# B&R Automation Studio project ROS_0101a
Automation Studio 4.5.2.102; technology packages: Acp10Arnc0 5.4.1, mappView 5.4.2

## Configuration ARsim

CPU PC_any, AutomationRuntime D4.52, Build 4.1.2, Vc V4.52.0

### Task classes (Cpu.sw)
```
Cyclic#1 (cycle 2000 us, tolerance 0 us):
  main <- Programs.main.prg
  rrbotctrl <- Programs.rrbotctrl.prg
Cyclic#8 (cycle 2000 us, tolerance 0 us):
  ros <- Programs.ros.prg
DataObjects: Acp10sys
NcDataObjects: acp10etxen <- MotionObjects.acp10etxen.dob, gConveyora <- MotionObjects.gConveyora.dob, gConveyori <- MotionObjects.gConveyori.dob, gRRBotJ1a <- gRRBotJ1obj.gRRBotJ1a.dob, gRRBotJ1i <- gRRBotJ1obj.gRRBotJ1i.dob, gRRBotJ2a <- gRRBotJ2obj.gRRBotJ2a.dob, gRRBotJ2i <- gRRBotJ2obj.gRRBotJ2i.dob
Binaries: udbdef, TCData, TCLang, arsvcreg, mvLoader, RRBot, ashwd, User, asfw, arconfig, sysconf, Role, ashwac, iomap, Conveyor, TC, OpcUaMap, acp10cfg, Acp10map
Libraries: operator, runtime, astime, AsIecCon, AsTCP, AsBrStr, AsICMP, RosNode, RosWrap, Acp10man, Acp10par, NcGlobal, Acp10sim, Acp10_MC, brsystem, sys_lib, MpAxis, MpCom, MpBase, standard, fileio, powerlnk, dataobj
```

### Hardware
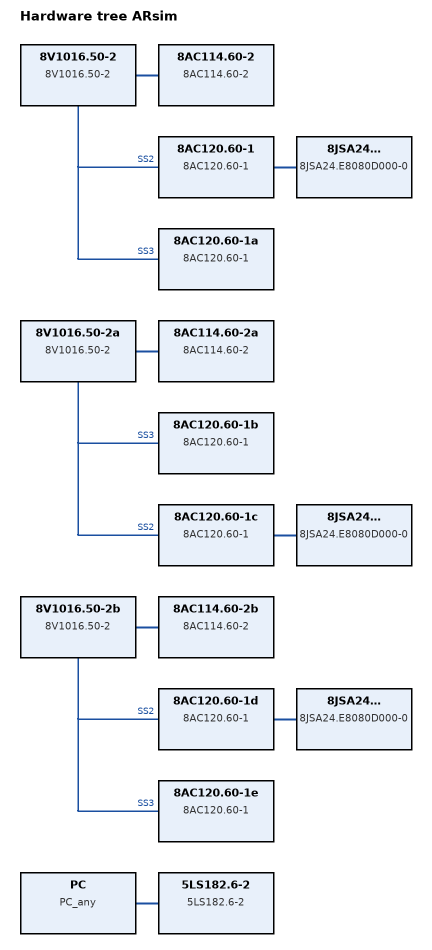
```
5LS182.6-2 : 5LS182.6-2 v1.3.1.0  [SL -> PC.SL1]
8AC114.60-2 : 8AC114.60-2 v1.0.0.8  [SS -> 8V1016.50-2.SS1; PLK1 -> 5LS182.6-2.IF1 [Cable Type=PowerlinkCable, Length=10, Version=1.0.0.2]; PLK2 -> 8AC114.60-2a.PLK1 [Cable Type=PowerlinkCable, Length=10, Version=1.0.0.2]]
8AC114.60-2a : 8AC114.60-2 v1.0.0.8  [SS -> 8V1016.50-2a.SS1; PLK1 -> 8AC114.60-2.PLK2 [Cable Type=PowerlinkCable, Length=10, Version=1.0.0.2]; PLK2 -> 8AC114.60-2b.PLK1 [Cable Type=PowerlinkCable, Length=10, Version=1.0.0.2]]
8AC114.60-2b : 8AC114.60-2 v1.0.0.8  [SS -> 8V1016.50-2b.SS1; PLK1 -> 8AC114.60-2a.PLK2 [Cable Type=PowerlinkCable, Length=10, Version=1.0.0.2]]
8AC120.60-1 : 8AC120.60-1 v2.2.0.0  [SS -> 8V1016.50-2.SS2]
8AC120.60-1a : 8AC120.60-1 v2.2.0.0  [SS -> 8V1016.50-2.SS3]
8AC120.60-1b : 8AC120.60-1 v2.2.0.0  [SS -> 8V1016.50-2a.SS3]
8AC120.60-1c : 8AC120.60-1 v2.2.0.0  [SS -> 8V1016.50-2a.SS2]
8AC120.60-1d : 8AC120.60-1 v2.2.0.0  [SS -> 8V1016.50-2b.SS2]
8AC120.60-1e : 8AC120.60-1 v2.2.0.0  [SS -> 8V1016.50-2b.SS3]
8JSA24.E8080D000-0 : 8JSA24.E8080D000-0 v1.0.6.30  [EC -> 8AC120.60-1.EC; MT -> 8V1016.50-2.MT1]
8JSA24.E8080D000-0a : 8JSA24.E8080D000-0 v1.0.6.30  [EC -> 8AC120.60-1c.EC; MT -> 8V1016.50-2a.MT1]
8JSA24.E8080D000-0b : 8JSA24.E8080D000-0 v1.0.6.30  [EC -> 8AC120.60-1d.EC; MT -> 8V1016.50-2b.MT1]
8V1016.50-2 : 8V1016.50-2 v2.2.0.0
  MotionTP = Acp10Arnc0
  Simulate = standard
  ActiveMotorSimulation_r1 = on
  BothEndSwitchesAreNormallyOpen_r1 = on
  QuickStopIsNormallyOpen_r1 = on
8V1016.50-2a : 8V1016.50-2 v2.2.0.0
  MotionTP = Acp10Arnc0
  Simulate = standard
  ActiveMotorSimulation_r1 = on
  BothEndSwitchesAreNormallyOpen_r1 = on
  QuickStopIsNormallyOpen_r1 = on
8V1016.50-2b : 8V1016.50-2 v2.2.0.0
  MotionTP = Acp10Arnc0
  Simulate = standard
  ActiveMotorSimulation_r1 = on
  BothEndSwitchesAreNormallyOpen_r1 = on
  QuickStopIsNormallyOpen_r1 = on
PC : PC_any v1.1.0.0 (OrderNumber=PC)
  Connector IF3:
    InternetAddress = 10.10.10.1
  ConfigurationID = ROS_0101a_ARsim
  SystemTick = 2000
  TaskClassIdleTime = 10000
  Cyclic1Duration = 2000
  Cyclic1Tolerance = 0
  Cyclic1Stack = 65535
  Cyclic2Duration = 20000
  Cyclic2Tolerance = 20000
  Cyclic8Duration = 2000
  Cyclic8Tolerance = 0
  Cyclic8Stack = 65535
  ActivateOpcUa = 1
  OpcUaInformationModels_PV_Version = 1
```

### Acp10cfg.ncc - PC/Motion/Acp10cfg.ncc
```
NcConfiguration (Version=5.04.1, NcSwId=Acp10)
  ACP10CF1_typ:
    cnt_nettrc_rec_drive = 1500
    bufsize_trace_upload = 1200
    tc_nc_man_task = Cyclic #1
    glob_pv_as_ncobject = Yes
    ncsys_dl_broadcast = Yes
    ncsys_dl_acp_reset = Yes
    safemc_log_err_to_ax = Yes
    network_init:
      ncsw_init_execute = Yes
      automatic_execute = No
      node_nr_warning = Yes
      net_err_before_ncact = Yes
    nettrc:
      enter_parsecrec = Yes
      enter_ncaction = Yes
      save_ring_startidx = Yes
    cam_prof_download:
      cam_dat_dl_parallel = No
      tc_cam_dl_parallel = Task class for NC Manager task
    plk_if[0]:
      if_name = SL1.IF1
      tc_CycDat_PLCopen = Task class for NC Manager task
      mc_broadcast_extdat = No
```

### Acp10map.ncm - PC/Motion/Acp10map.ncm
```
NcMapping (NcSwId=Acp10, DisabledNodesAreHidden=False)
  NcObject gConveyor (ModuleId=8V1016.50-2, Type=ncAXIS, Channel=1, AcoposSimulation=Standard, InitParameter=gConveyori, AcoposParameter=gConveyora, Disabled=FALSE, ModuleDisabled=FALSE)
  NcObject 8V1016.50-2_ncV_AXIS1 (ModuleId=8V1016.50-2, Type=ncV_AXIS, Channel=1, Disabled=TRUE, ModuleDisabled=FALSE)
  NcObject gRRBotJ1 (ModuleId=8V1016.50-2a, Type=ncAXIS, Channel=1, AcoposSimulation=Off, InitParameter=gRRBotJ1i, AcoposParameter=gRRBotJ1a, Disabled=FALSE, ModuleDisabled=FALSE)
  NcObject 8V1016.50-2a_ncV_AXIS1 (ModuleId=8V1016.50-2a, Type=ncV_AXIS, Channel=1, Disabled=TRUE, ModuleDisabled=FALSE)
  NcObject gRRBotJ2 (ModuleId=8V1016.50-2b, Type=ncAXIS, Channel=1, AcoposSimulation=Off, InitParameter=gRRBotJ2i, AcoposParameter=gRRBotJ2a, Disabled=FALSE, ModuleDisabled=FALSE)
  NcObject 8V1016.50-2b_ncV_AXIS1 (ModuleId=8V1016.50-2b, Type=ncV_AXIS, Channel=1, Disabled=TRUE, ModuleDisabled=FALSE)
```

### Conveyor.mpaxisbasic - PC/Motion/Conveyor.mpaxisbasic
```
Element gMpLinkConveyor (Type=mpaxisbasic)
  AxisConfiguration = AxisWithConfiguration
    Axis:
      BaseType = 4
      MeasurementUnit = 2
      MeasurementResolution = 0.001
      SoftwareLimitPositions:
        LowerLimit = -100
        UpperLimit = 100
      PeriodSettings:
        Period = 0
      MovementLimits:
        VelocityPositive = 10
        VelocityNegative = 10
        Acceleration = 50
        Deceleration = 50
    Drive:
      Transformation:
        ReferenceDistance = 1
      Controller:
        LoopFilters:
          [0]
          [1]
          [2]
  Alarms = MpAlarmX
```

### RRBot.mpaxisbasic - PC/Motion/RRBot.mpaxisbasic
```
Element gMpLinkRRBotJ1 (Type=mpaxisbasic)
  AxisConfiguration = AxisWithConfiguration
    Axis:
      MeasurementUnit = 2
      MeasurementResolution = 0.001
      SoftwareLimitPositions:
        LowerLimit = -100
        UpperLimit = 100
      PeriodSettings:
        Period = 360
      MovementLimits:
        VelocityPositive = 3600
        VelocityNegative = 3600
        Acceleration = 36000
        Deceleration = 36000
    Drive:
      Transformation:
        ReferenceDistance = 1
      Controller:
        LoopFilters:
          [0]
          [1]
          [2]
  Alarms = MpAlarmX
Element gMpLinkRRBotJ2 (Type=mpaxisbasic)
  AxisConfiguration = AxisWithConfiguration
    Axis:
      MeasurementUnit = 2
      MeasurementResolution = 0.001
      SoftwareLimitPositions:
        LowerLimit = -100
        UpperLimit = 100
      PeriodSettings:
        Period = 360
      MovementLimits:
        VelocityPositive = 3600
        VelocityNegative = 3600
        Acceleration = 36000
        Deceleration = 36000
    Drive:
      Transformation:
        ReferenceDistance = 1
      Controller:
        LoopFilters:
          [0]
          [1]
          [2]
  Alarms = MpAlarmX
```

## Logical view

Binary libraries used (declarations not repeated): operator, runtime, astime, AsIecCon, AsTCP, AsBrStr, AsICMP, brsystem, sys_lib, MpCom 5.04.2, standard, MpAxis 1.67.0, MpBase 5.04.1, NcGlobal 5.04.1, Acp10_MC 5.04.1, Acp10man 5.04.1, Acp10par 5.04.1, Acp10sim 5.04.1

### Global.var - Global variables
```iecst
VAR
	joint2PositionDegrees : REAL;
	joint1PositionDegrees : REAL;
	joint1ActualPosition : REAL;
	joint2ActualPosition : REAL;
	joint2SetPosition : REAL;
	joint1SetPosition : REAL;
	redCaseComplete : BOOL;
	greenCaseComplete : BOOL;
	blueCaseComplete : BOOL;
	speakNow : BOOL;
	textCommand : STRING[1000];
	wakeCommand : BOOL;
	TestVar : USINT;
	command : USINT;
	ROSCommand : RosWrapper_FulfilledCommand_Type;
	gConveyor : ACP10AXIS_typ;
	gRRBotJ1 : ACP10AXIS_typ;
	gRRBotJ2 : ACP10AXIS_typ;
END_VAR
```

### Package Logical/Libraries - Global libraries

### Library Logical/Libraries/RosNode (ANSIC)

#### rosnode.cpp - Init, cyclic, exit code
```cpp
#include "rosnode.hpp"

// Constructor
RosNode::RosNode()
{
	_nh.initNode();
	_nh.setSpinTimeout(1);
}

// Destructor
RosNode::~RosNode()
{
}

// Message callback for the fulfilledCommand subscription
voice_interaction_robot_msgs::FulfilledVoiceCommand messageCallback( const voice_interaction_robot_msgs::FulfilledVoiceCommand& fulfilledCommand)
{
	return fulfilledCommand;
}

// Cyclic execution logic
voice_interaction_robot_msgs::FulfilledVoiceCommand RosNode::Cyclic(std_msgs::String wakeWord, BOOL wakeCommand)
{
	// Create my publisher
	static ros::Publisher control("/wake_word", &wakeWord);

	// Create my subscriber
	static ros::Subscriber<voice_interaction_robot_msgs::FulfilledVoiceCommand> status("/voice_interaction_node/fulfilled_command", messageCallback);

	// Initialization logic for publishers and subscribers
	if (!_init)
	{
		_nh.advertise(control);
		_nh.subscribe(status);
		_init = true;
	}

	// We only publish the wakeWord if commanded to do so (i.e. not cyclic publishing)
	if (wakeCommand == true)
	control.publish( &wakeWord);

	// This call runs all of the underlying node's cyclic logic.
	_nh.spinOnce();

	// Keeping track of new data received on the callback function, and returning this data
	if (status.callbackCounter_ != _oldCallbackCounter)
	{
		_oldCallbackCounter = status.callbackCounter_;
		return status.fulfilledCommand_;
	} else
	{
	_oldCallbackCounter = status.callbackCounter_;
	voice_interaction_robot_msgs::FulfilledVoiceCommand dummyMessage;
	brsmemset((UDINT)&dummyMessage,0,sizeof(dummyMessage));
	return dummyMessage;
	}
};
```

#### rosnode.hpp
```cpp
#include "hardware.h"

// This is where we include references to all custom message packages
#include "ros/node_handle.h"
#include "std_msgs/String.h"
#include "geometry_msgs/Twist.h"
#include "sound_play/SoundRequest.h"
#include "voice_interaction_robot_msgs/FulfilledVoiceCommand.h"

class RosNode
{
	public:
		// Constructor and destructor
		RosNode();
		virtual ~RosNode();
		// Cyclic function for processing all logic
		voice_interaction_robot_msgs::FulfilledVoiceCommand Cyclic(std_msgs::String wakeWord, BOOL wakeCommand);

	private:
		// Create the node handle
		ros::NodeHandle_<Hardware> _nh;

		// Defining several local PVs
		BOOL _init;
		UDINT _oldCallbackCounter;
};
```

#### hardware.h
```c
#include <bur/plctypes.h>

#ifdef _DEFAULT_INCLUDES
#include <AsDefault.h>
#endif

class Hardware
{
	public:
	Hardware()
	{
		// Initializing all variables (otherwise they can have random values)
		_programStartTime = clock_ms();
		_step = 0;
		_ident = 0;
		_recvData = 0;
		_lastError = 0;
		_errorFlag = false;
		_recvTimeout = 0;
		brsmemset(reinterpret_cast<UDINT>(&_tcpOpen),0,sizeof(_tcpOpen));
		brsmemset(reinterpret_cast<UDINT>(&_tcpClient),0,sizeof(_tcpClient));
		brsmemset(reinterpret_cast<UDINT>(&_tcpRecv),0,sizeof(_tcpRecv));
		brsmemset(reinterpret_cast<UDINT>(&_tcpSend),0,sizeof(_tcpSend));
		brsmemset(reinterpret_cast<UDINT>(&_tcpClose),0,sizeof(_tcpClose));
	}

	// any initialization code necessary to use the serial port
	void init()
	{
		// we need to stay in this method until we've successfully connected, hence the while loop
		while (_step < 3) // STEP_CONNECTED
		{
			switch (_step)
			{
				case 0: // STEP_START
					initData();
					_step = 1; // STEP_OPEN_SOCKET
					break;

				/* opens ethernet interface for use with SSL */
				case 1: // STEP_OPEN_SOCKET
					openSocket();
					break;

				/* connects to the server */
				case 2: // STEP_CONNECT_TO_SERVER
					connectToServer();
					break;

				/* holding state once we're connected */
				case 3: // STEP_CONNECTED
					break;
			}
		}
	}

	// read a byte from the serial port. -1 = failure
	int read()
	{
		return receiveData();
	}

	// write data to the connection to ROS
	void write(USINT* data, int length)
	{
		sendData(data, length);
	}

	// returns milliseconds since start of program
	unsigned long time()
	{
		return (long) DiffT(clock_ms(),_programStartTime);
	}

	UDINT getLoopCounter()
	{
		return _loopCounter;
	}

	private:

	void initData()
	{
		/***** internal parameter assignments for all FBs *****/
		// TCP open FB
		_tcpOpen.pIfAddr 	= 0;
		_tcpOpen.port 		= 0;
		_tcpOpen.options 	= tcpOPT_REUSEADDR;

		// TCP client FB
		_tcpClient.portserv = 11411;
		_tcpClient.pServer  = (UDINT) "192.168.56.101";

		// TCP receive FB
		_tcpRecv.pData   = (UDINT) &(_recvData);
		_tcpRecv.datamax = sizeof(_recvData);
		_tcpRecv.flags   = 0;

		// TCP send FB
		_tcpSend.flags   = 0;
	}

	/* Opens a socket with the given port. */
	void openSocket()
	{
		_tcpOpen.enable = 1;

		TcpOpen(&_tcpOpen);

		if (_tcpOpen.status == ERR_OK)
		{
			_step 	  = 2; // STEP_CONNECT_TO_SERVER
			_ident 	  = _tcpOpen.ident;
		}
		else if (_tcpOpen.status != ERR_FUB_BUSY )
		{
			_step	  = 500; // STEP_ERROR
			_lastError = _tcpOpen.status;
		}
	}

	/* Connects to the given server. */
	void connectToServer()
	{
		_tcpClient.enable   = 1;
		_tcpClient.ident 	  = _ident;
		TcpClient(&_tcpClient);

		if (_tcpClient.status == ERR_OK)
		{
			_step = 3; // STEP_CONNECTED
		}
		else if (_tcpClient.status != ERR_FUB_BUSY)
		{
			_errorFlag = true;
			_step 	  = 6; // STEP_CLOSE_SOCKET
			_lastError = _tcpClient.status;
		}
	}

	/* Receives data from server. */
	INT receiveData()
	{
		_tcpRecv.enable  = 1;
		_tcpRecv.ident   = _ident;
		while ((_tcpRecv.status == ERR_FUB_ENABLE_FALSE) || (_tcpRecv.status == ERR_FUB_BUSY))
		{
			TcpRecv(&_tcpRecv);
		}

		if (_tcpRecv.status == ERR_OK)
		{
			_recvTimeout = 0;
			_tcpRecv.enable = false;
			TcpRecv(&_tcpRecv);
			return _recvData;
		}
		else if (_tcpRecv.status == tcpERR_NO_DATA) 					/* no data received - try again */
		{
			_recvTimeout 	   = _recvTimeout + 1;
			_tcpRecv.enable = false;
			TcpRecv(&_tcpRecv);
			return -1;
		}
		else if (_tcpRecv.status == ERR_FUB_BUSY)
		{
			return -1;
		}
		else // we have an error
		{
			_errorFlag = true;
			_step 	  = 6; // STEP_CLOSE_SOCKET
			_lastError = _tcpSend.status;
			_tcpRecv.enable = false;
			TcpRecv(&_tcpRecv);
			return -1;
		}
	}

	/* Sends data to the server */
	void sendData(USINT* data, int length)
	{
		_tcpSend.enable  = 1;
		_tcpSend.ident   = _ident;
		_tcpSend.pData   = (UDINT) data;
		_tcpSend.datalen = (UDINT) length;
		TcpSend(&_tcpSend);
		while ((_tcpSend.status == ERR_FUB_BUSY) || (_tcpSend.status == ERR_FUB_ENABLE_FALSE))
		{
			TcpSend(&_tcpSend);
		}

		if (_tcpSend.status == ERR_OK)
		{
			_tcpSend.enable = false;
			TcpSend(&_tcpSend);
			_step = 5; // STEP_RECEIVE_DATA
			return;
		}
		else if (_tcpSend.status != ERR_FUB_BUSY)
		{
			_tcpSend.enable = false;
			TcpSend(&_tcpSend);
			_errorFlag = true;
			_step	  = 6; // STEP_CLOSE_SOCKET
			_lastError = _tcpSend.status;
			return;
		}
	}

	UDINT _programStartTime;
	UINT _step;
	UDINT _ident;
	USINT _recvData;
	UINT _lastError;
	BOOL _errorFlag;
	UDINT _recvTimeout;
	UDINT _loopCounter;
	TcpOpen_typ _tcpOpen;
	TcpClient_typ _tcpClient;
	TcpRecv_typ _tcpRecv;
	TcpSend_typ _tcpSend;
	TcpClose_typ _tcpClose;
};
```

#### Time.h
```c
#ifndef _ROS_std_msgs_Time_h
#define _ROS_std_msgs_Time_h

#include <stdint.h>
#include <string.h>
#include <stdlib.h>
#include "../ros/msg.h"
#include "../ros/time.h"

namespace std_msgs
{

  class Time : public ros::Msg
  {
    public:
      typedef ros::Time _data_type;
      _data_type data;

    Time():
      data()
    {
    }

    virtual int serialize(unsigned char *outbuffer) const
    {
      int offset = 0;
      *(outbuffer + offset + 0) = (this->data.sec >> (8 * 0)) & 0xFF;
      *(outbuffer + offset + 1) = (this->data.sec >> (8 * 1)) & 0xFF;
      *(outbuffer + offset + 2) = (this->data.sec >> (8 * 2)) & 0xFF;
      *(outbuffer + offset + 3) = (this->data.sec >> (8 * 3)) & 0xFF;
      offset += sizeof(this->data.sec);
      *(outbuffer + offset + 0) = (this->data.nsec >> (8 * 0)) & 0xFF;
      *(outbuffer + offset + 1) = (this->data.nsec >> (8 * 1)) & 0xFF;
      *(outbuffer + offset + 2) = (this->data.nsec >> (8 * 2)) & 0xFF;
      *(outbuffer + offset + 3) = (this->data.nsec >> (8 * 3)) & 0xFF;
      offset += sizeof(this->data.nsec);
      return offset;
    }

    virtual int deserialize(unsigned char *inbuffer)
    {
      int offset = 0;
      this->data.sec =  ((uint32_t) (*(inbuffer + offset)));
      this->data.sec |= ((uint32_t) (*(inbuffer + offset + 1))) << (8 * 1);
      this->data.sec |= ((uint32_t) (*(inbuffer + offset + 2))) << (8 * 2);
      this->data.sec |= ((uint32_t) (*(inbuffer + offset + 3))) << (8 * 3);
      offset += sizeof(this->data.sec);
      this->data.nsec =  ((uint32_t) (*(inbuffer + offset)));
      this->data.nsec |= ((uint32_t) (*(inbuffer + offset + 1))) << (8 * 1);
      this->data.nsec |= ((uint32_t) (*(inbuffer + offset + 2))) << (8 * 2);
      this->data.nsec |= ((uint32_t) (*(inbuffer + offset + 3))) << (8 * 3);
      offset += sizeof(this->data.nsec);
     return offset;
    }

    const char * getType(){ return "std_msgs/Time"; };
    const char * getMD5(){ return "cd7166c74c552c311fbcc2fe5a7bc289"; };

  };

}
#endif
```

#### String.h
```c
#ifndef _ROS_std_msgs_String_h
#define _ROS_std_msgs_String_h

#include <stdint.h>
#include <string.h>
#include <stdlib.h>
#include "../ros/msg.h"

namespace std_msgs
{

  class String : public ros::Msg
  {
    public:
      typedef const char* _data_type;
      _data_type data;

    String():
      data("")
    {
    }

    virtual int serialize(unsigned char *outbuffer) const
    {
      int offset = 0;
      uint32_t length_data = strlen(this->data);
      varToArr(outbuffer + offset, length_data);
      offset += 4;
      memcpy(outbuffer + offset, this->data, length_data);
      offset += length_data;
      return offset;
    }

    virtual int deserialize(unsigned char *inbuffer)
    {
      int offset = 0;
      uint32_t length_data;
      arrToVar(length_data, (inbuffer + offset));
      offset += 4;
      for(unsigned int k= offset; k< offset+length_data; ++k){
          inbuffer[k-1]=inbuffer[k];
      }
      inbuffer[offset+length_data-1]=0;
      this->data = (char *)(inbuffer + offset-1);
      offset += length_data;
     return offset;
    }

    const char * getType(){ return "std_msgs/String"; };
    const char * getMD5(){ return "992ce8a1687cec8c8bd883ec73ca41d1"; };

  };

}
#endif
```

#### publisher.h
```c
/*
 * Software License Agreement (BSD License)
 *
 * Copyright (c) 2011, Willow Garage, Inc.
 * All rights reserved.
 *
 * Redistribution and use in source and binary forms, with or without
 * modification, are permitted provided that the following conditions
 * are met:
 *
 *  * Redistributions of source code must retain the above copyright
 *    notice, this list of conditions and the following disclaimer.
 *  * Redistributions in binary form must reproduce the above
 *    copyright notice, this list of conditions and the following
 *    disclaimer in the documentation and/or other materials provided
 *    with the distribution.
 *  * Neither the name of Willow Garage, Inc. nor the names of its
 *    contributors may be used to endorse or promote prducts derived
 *    from this software without specific prior written permission.
 *
 * THIS SOFTWARE IS PROVIDED BY THE COPYRIGHT HOLDERS AND CONTRIBUTORS
 * "AS IS" AND ANY EXPRESS OR IMPLIED WARRANTIES, INCLUDING, BUT NOT
 * LIMITED TO, THE IMPLIED WARRANTIES OF MERCHANTABILITY AND FITNESS
 * FOR A PARTICULAR PURPOSE ARE DISCLAIMED. IN NO EVENT SHALL THE
 * COPYRIGHT OWNER OR CONTRIBUTORS BE LIABLE FOR ANY DIRECT, INDIRECT,
 * INCIDENTAL, SPECIAL, EXEMPLARY, OR CONSEQUENTIAL DAMAGES (INCLUDING,
 * BUT NOT LIMITED TO, PROCUREMENT OF SUBSTITUTE GOODS OR SERVICES;
 * LOSS OF USE, DATA, OR PROFITS; OR BUSINESS INTERRUPTION) HOWEVER
 * CAUSED AND ON ANY THEORY OF LIABILITY, WHETHER IN CONTRACT, STRICT
 * LIABILITY, OR TORT (INCLUDING NEGLIGENCE OR OTHERWISE) ARISING IN
 * ANY WAY OUT OF THE USE OF THIS SOFTWARE, EVEN IF ADVISED OF THE
 * POSSIBILITY OF SUCH DAMAGE.
 */

#ifndef _ROS_PUBLISHER_H_
#define _ROS_PUBLISHER_H_

#include "../rosserial_msgs/TopicInfo.h"
#include "../ros/node_handle.h"

namespace ros
{

/* Generic Publisher */
class Publisher
{
public:
  Publisher(const char * topic_name, Msg * msg, int endpoint = rosserial_msgs::TopicInfo::ID_PUBLISHER) :
    topic_(topic_name),
    msg_(msg),
    endpoint_(endpoint) {};

  int publish(const Msg * msg)
  {
    return nh_->publish(id_, msg);
  };
  int getEndpointType()
  {
    return endpoint_;
  }

  const char * topic_;
  Msg *msg_;
  // id_ and no_ are set by NodeHandle when we advertise
  int id_;
  NodeHandleBase_* nh_;

private:
  int endpoint_;
};

}

#endif
```

#### node_handle.h
```c
/*
 * Software License Agreement (BSD License)
 *
 * Copyright (c) 2011, Willow Garage, Inc.
 * All rights reserved.
 *
 * Redistribution and use in source and binary forms, with or without
 * modification, are permitted provided that the following conditions
 * are met:
 *
 *  * Redistributions of source code must retain the above copyright
 *    notice, this list of conditions and the following disclaimer.
 *  * Redistributions in binary form must reproduce the above
 *    copyright notice, this list of conditions and the following
 *    disclaimer in the documentation and/or other materials provided
 *    with the distribution.
 *  * Neither the name of Willow Garage, Inc. nor the names of its
 *    contributors may be used to endorse or promote prducts derived
 *    from this software without specific prior written permission.
 *
 * THIS SOFTWARE IS PROVIDED BY THE COPYRIGHT HOLDERS AND CONTRIBUTORS
 * "AS IS" AND ANY EXPRESS OR IMPLIED WARRANTIES, INCLUDING, BUT NOT
 * LIMITED TO, THE IMPLIED WARRANTIES OF MERCHANTABILITY AND FITNESS
 * FOR A PARTICULAR PURPOSE ARE DISCLAIMED. IN NO EVENT SHALL THE
 * COPYRIGHT OWNER OR CONTRIBUTORS BE LIABLE FOR ANY DIRECT, INDIRECT,
 * INCIDENTAL, SPECIAL, EXEMPLARY, OR CONSEQUENTIAL DAMAGES (INCLUDING,
 * BUT NOT LIMITED TO, PROCUREMENT OF SUBSTITUTE GOODS OR SERVICES;
 * LOSS OF USE, DATA, OR PROFITS; OR BUSINESS INTERRUPTION) HOWEVER
 * CAUSED AND ON ANY THEORY OF LIABILITY, WHETHER IN CONTRACT, STRICT
 * LIABILITY, OR TORT (INCLUDING NEGLIGENCE OR OTHERWISE) ARISING IN
 * ANY WAY OUT OF THE USE OF THIS SOFTWARE, EVEN IF ADVISED OF THE
 * POSSIBILITY OF SUCH DAMAGE.
 */

#ifndef ROS_NODE_HANDLE_H_
#define ROS_NODE_HANDLE_H_

#include <stdint.h>

#include "../std_msgs/Time.h"
#include "../rosserial_msgs/TopicInfo.h"
#include "../rosserial_msgs/Log.h"
#include "../rosserial_msgs/RequestParam.h"

#include "../ros/msg.h"

namespace ros
{

class NodeHandleBase_
{
public:
  virtual int publish(int id, const Msg* msg) = 0;
  virtual int spinOnce() = 0;
  virtual bool connected() = 0;
};
}

#include "../ros/publisher.h"
#include "../ros/subscriber.h"
#include "../ros/service_server.h"
#include "../ros/service_client.h"

namespace ros
{

const int SPIN_OK = 0;
const int SPIN_ERR = -1;
const int SPIN_TIMEOUT = -2;
const int SPIN_TIMEOUT2 = -3;

const uint8_t SYNC_SECONDS  = 5;
const uint8_t MODE_FIRST_FF = 0;
/*
 * The second sync byte is a protocol version. It's value is 0xff for the first
 * version of the rosserial protocol (used up to hydro), 0xfe for the second version
 * (introduced in hydro), 0xfd for the next, and so on. Its purpose is to enable
 * detection of mismatched protocol versions (e.g. hydro rosserial_python with groovy
 * rosserial_arduino. It must be changed in both this file and in
 * rosserial_python/src/rosserial_python/SerialClient.py
 */
const uint8_t MODE_PROTOCOL_VER   = 1;
const uint8_t PROTOCOL_VER1       = 0xff; // through groovy
const uint8_t PROTOCOL_VER2       = 0xfe; // in hydro
const uint8_t PROTOCOL_VER        = PROTOCOL_VER2;
const uint8_t MODE_SIZE_L         = 2;
const uint8_t MODE_SIZE_H         = 3;
const uint8_t MODE_SIZE_CHECKSUM  = 4;    // checksum for msg size received from size L and H
const uint8_t MODE_TOPIC_L        = 5;    // waiting for topic id
const uint8_t MODE_TOPIC_H        = 6;
const uint8_t MODE_MESSAGE        = 7;
const uint8_t MODE_MSG_CHECKSUM   = 8;    // checksum for msg and topic id

const uint8_t SERIAL_MSG_TIMEOUT  = 20;   // 20 milliseconds to recieve all of message data

using rosserial_msgs::TopicInfo;

/* Node Handle */
template<class Hardware,
         int MAX_SUBSCRIBERS = 25,
         int MAX_PUBLISHERS = 25,
         int INPUT_SIZE = 512,
         int OUTPUT_SIZE = 512>
class NodeHandle_ : public NodeHandleBase_
{
protected:
  Hardware hardware_;

  /* time used for syncing */
  uint32_t rt_time;

  /* used for computing current time */
  uint32_t sec_offset, nsec_offset;

  /* Spinonce maximum work timeout */
  uint32_t spin_timeout_;

  uint8_t message_in[INPUT_SIZE];
  uint8_t message_out[OUTPUT_SIZE];

  Publisher * publishers[MAX_PUBLISHERS];
  Subscriber_ * subscribers[MAX_SUBSCRIBERS];

  /*
   * Setup Functions
   */
public:
  NodeHandle_() : configured_(false)
  {

    for (unsigned int i = 0; i < MAX_PUBLISHERS; i++)
      publishers[i] = 0;

    for (unsigned int i = 0; i < MAX_SUBSCRIBERS; i++)
      subscribers[i] = 0;

    for (unsigned int i = 0; i < INPUT_SIZE; i++)
      message_in[i] = 0;

    for (unsigned int i = 0; i < OUTPUT_SIZE; i++)
      message_out[i] = 0;

    req_param_resp.ints_length = 0;
    req_param_resp.ints = NULL;
    req_param_resp.floats_length = 0;
    req_param_resp.floats = NULL;
    req_param_resp.ints_length = 0;
    req_param_resp.ints = NULL;

    spin_timeout_ = 0;
  }

  Hardware* getHardware()
  {
    return &hardware_;
  }

  /* Start serial, initialize buffers */
  void initNode()
  {
    hardware_.init();
    mode_ = 0;
    bytes_ = 0;
    index_ = 0;
    topic_ = 0;
  };

  /* Start a named port, which may be network server IP, initialize buffers */
  void initNode(char *portName)
  {
    hardware_.init(portName);
    mode_ = 0;
    bytes_ = 0;
    index_ = 0;
    topic_ = 0;
  };

  /**
   * @brief Sets the maximum time in millisconds that spinOnce() can work.
   * This will not effect the processing of the buffer, as spinOnce processes
   * one byte at a time. It simply sets the maximum time that one call can
   * process for. You can choose to clear the buffer if that is beneficial if
   * SPIN_TIMEOUT is returned from spinOnce().
   * @param timeout The timeout in milliseconds that spinOnce will function.
   */
  void setSpinTimeout(const uint32_t& timeout)
  {
     spin_timeout_ = timeout;
  }

protected:
  //State machine variables for spinOnce
  int mode_;
  int bytes_;
  int topic_;
  int index_;
  int checksum_;

  bool configured_;

  /* used for syncing the time */
  uint32_t last_sync_time;
  uint32_t last_sync_receive_time;
  uint32_t last_msg_timeout_time;

public:
  /* This function goes in your loop() function, it handles
   *  serial input and callbacks for subscribers.
   */
  virtual int spinOnce()
  {
    /* restart if timed out */
    uint32_t c_time = hardware_.time();
    if ((c_time - last_sync_receive_time) > (SYNC_SECONDS * 2200))
    {
      configured_ = false;
    }

    /* reset if message has timed out */
    if (mode_ != MODE_FIRST_FF)
    {
      if (c_time > last_msg_timeout_time)
      {
        mode_ = MODE_FIRST_FF;
      }
    }

    /* while available buffer, read data */
    while (true)
    {
      // If a timeout has been specified, check how long spinOnce has been running.
      if (spin_timeout_ > 0)
      {
        // If the maximum processing timeout has been exceeded, exit with error.
        // The next spinOnce can continue where it left off, or optionally
        // based on the application in use, the hardware buffer could be flushed
        // and start fresh.
        if ((hardware_.time() - c_time) > spin_timeout_)
        {
          // Exit the spin, processing timeout exceeded.
          return SPIN_TIMEOUT;
        }
      }
      int data = hardware_.read();
      if (data < 0)
        break;
      checksum_ += data;
      if (mode_ == MODE_MESSAGE)          /* message data being recieved */
      {
        message_in[index_++] = data;
        bytes_--;
        if (bytes_ == 0)                 /* is message complete? if so, checksum */
          mode_ = MODE_MSG_CHECKSUM;
      }
      else if (mode_ == MODE_FIRST_FF)
      {
        if (data == 0xff)
        {
          mode_++;
          last_msg_timeout_time = c_time + SERIAL_MSG_TIMEOUT;
        }
        else if (hardware_.time() - c_time > (SYNC_SECONDS * 1000))
        {
          /* We have been stuck in spinOnce too long, return error */
          configured_ = false;
          return SPIN_TIMEOUT;
        }
      }
      else if (mode_ == MODE_PROTOCOL_VER)
      {
        if (data == PROTOCOL_VER)
        {
          mode_++;
        }
        else
        {
          mode_ = MODE_FIRST_FF;
          if (configured_ == false)
            requestSyncTime();  /* send a msg back showing our protocol version */
        }
      }
      else if (mode_ == MODE_SIZE_L)      /* bottom half of message size */
      {
        bytes_ = data;
        index_ = 0;
        mode_++;
        checksum_ = data;               /* first byte for calculating size checksum */
      }
      else if (mode_ == MODE_SIZE_H)      /* top half of message size */
      {
        bytes_ += data << 8;
        mode_++;
      }
      else if (mode_ == MODE_SIZE_CHECKSUM)
      {
        if ((checksum_ % 256) == 255)
          mode_++;
        else
          mode_ = MODE_FIRST_FF;          /* Abandon the frame if the msg len is wrong */
      }
      else if (mode_ == MODE_TOPIC_L)     /* bottom half of topic id */
      {
        topic_ = data;
        mode_++;
        checksum_ = data;               /* first byte included in checksum */
      }
      else if (mode_ == MODE_TOPIC_H)     /* top half of topic id */
      {
        topic_ += data << 8;
        mode_ = MODE_MESSAGE;
        if (bytes_ == 0)
          mode_ = MODE_MSG_CHECKSUM;
      }
      else if (mode_ == MODE_MSG_CHECKSUM)    /* do checksum */
      {
        mode_ = MODE_FIRST_FF;
        if ((checksum_ % 256) == 255)
        {
          if (topic_ == TopicInfo::ID_PUBLISHER)
          {
            requestSyncTime();
            negotiateTopics();
            last_sync_time = c_time;
            last_sync_receive_time = c_time;
            return SPIN_ERR;
          }
          else if (topic_ == TopicInfo::ID_TIME)
          {
            syncTime(message_in);
          }
          else if (topic_ == TopicInfo::ID_PARAMETER_REQUEST)
          {
            req_param_resp.deserialize(message_in);
            param_recieved = true;
          }
          else if (topic_ == TopicInfo::ID_TX_STOP)
          {
            configured_ = false;
          }
          else
          {
            if (subscribers[topic_ - 100])
              subscribers[topic_ - 100]->callback(message_in);
          }
        }
      }
    }

    /* occasionally sync time */
    if (configured_ && ((c_time - last_sync_time) > (SYNC_SECONDS * 500)))
    {
      requestSyncTime();
      last_sync_time = c_time;
    }

    return SPIN_OK;
  }

  /* Are we connected to the PC? */
  virtual bool connected()
  {
    return configured_;
  };

  /********************************************************************
   * Time functions
   */

  void requestSyncTime()
  {
    std_msgs::Time t;
    publish(TopicInfo::ID_TIME, &t);
    rt_time = hardware_.time();
  }

  void syncTime(uint8_t * data)
  {
    std_msgs::Time t;
    uint32_t offset = hardware_.time() - rt_time;

    t.deserialize(data);
    t.data.sec += offset / 1000;
    t.data.nsec += (offset % 1000) * 1000000UL;

    this->setNow(t.data);
    last_sync_receive_time = hardware_.time();
  }

  Time now()
  {
    uint32_t ms = hardware_.time();
    Time current_time;
    current_time.sec = ms / 1000 + sec_offset;
    current_time.nsec = (ms % 1000) * 1000000UL + nsec_offset;
    normalizeSecNSec(current_time.sec, current_time.nsec);
    return current_time;
  }

  void setNow(Time & new_now)
  {
    uint32_t ms = hardware_.time();
    sec_offset = new_now.sec - ms / 1000 - 1;
    nsec_offset = new_now.nsec - (ms % 1000) * 1000000UL + 1000000000UL;
    normalizeSecNSec(sec_offset, nsec_offset);
  }

  /********************************************************************
   * Topic Management
   */

  /* Register a new publisher */
  bool advertise(Publisher & p)
  {
    for (int i = 0; i < MAX_PUBLISHERS; i++)
    {
      if (publishers[i] == 0) // empty slot
      {
        publishers[i] = &p;
        p.id_ = i + 100 + MAX_SUBSCRIBERS;
        p.nh_ = this;
        return true;
      }
    }
    return false;
  }

  /* Register a new subscriber */
  template<typename SubscriberT>
  bool subscribe(SubscriberT& s)
  {
    for (int i = 0; i < MAX_SUBSCRIBERS; i++)
    {
      if (subscribers[i] == 0) // empty slot
      {
        subscribers[i] = static_cast<Subscriber_*>(&s);
        s.id_ = i + 100;
        return true;
      }
    }
    return false;
  }

  /* Register a new Service Server */
  template<typename MReq, typename MRes, typename ObjT>
  bool advertiseService(ServiceServer<MReq, MRes, ObjT>& srv)
  {
    bool v = advertise(srv.pub);
    for (int i = 0; i < MAX_SUBSCRIBERS; i++)
    {
      if (subscribers[i] == 0) // empty slot
      {
        subscribers[i] = static_cast<Subscriber_*>(&srv);
        srv.id_ = i + 100;
        return v;
      }
    }
    return false;
  }

  /* Register a new Service Client */
  template<typename MReq, typename MRes>
  bool serviceClient(ServiceClient<MReq, MRes>& srv)
  {
    bool v = advertise(srv.pub);
    for (int i = 0; i < MAX_SUBSCRIBERS; i++)
    {
      if (subscribers[i] == 0) // empty slot
      {
        subscribers[i] = static_cast<Subscriber_*>(&srv);
        srv.id_ = i + 100;
        return v;
      }
    }
    return false;
  }

  void negotiateTopics()
  {
    rosserial_msgs::TopicInfo ti;
    int i;
    for (i = 0; i < MAX_PUBLISHERS; i++)
    {
      if (publishers[i] != 0) // non-empty slot
      {
        ti.topic_id = publishers[i]->id_;
        ti.topic_name = (char *) publishers[i]->topic_;
        ti.message_type = (char *) publishers[i]->msg_->getType();
        ti.md5sum = (char *) publishers[i]->msg_->getMD5();
        ti.buffer_size = OUTPUT_SIZE;
        publish(publishers[i]->getEndpointType(), &ti);
      }
    }
    for (i = 0; i < MAX_SUBSCRIBERS; i++)
    {
      if (subscribers[i] != 0) // non-empty slot
      {
        ti.topic_id = subscribers[i]->id_;
        ti.topic_name = (char *) subscribers[i]->topic_;
        ti.message_type = (char *) subscribers[i]->getMsgType();
        ti.md5sum = (char *) subscribers[i]->getMsgMD5();
        ti.buffer_size = INPUT_SIZE;
        publish(subscribers[i]->getEndpointType(), &ti);
      }
    }
    configured_ = true;
  }

  virtual int publish(int id, const Msg * msg)
  {
    if (id >= 100 && !configured_)
      return 0;

    /* serialize message */
    int l = msg->serialize(message_out + 7);

    /* setup the header */
    message_out[0] = 0xff;
    message_out[1] = PROTOCOL_VER;
    message_out[2] = (uint8_t)((uint16_t)l & 255);
    message_out[3] = (uint8_t)((uint16_t)l >> 8);
    message_out[4] = 255 - ((message_out[2] + message_out[3]) % 256);
    message_out[5] = (uint8_t)((int16_t)id & 255);
    message_out[6] = (uint8_t)((int16_t)id >> 8);

    /* calculate checksum */
    int chk = 0;
    for (int i = 5; i < l + 7; i++)
      chk += message_out[i];
    l += 7;
    message_out[l++] = 255 - (chk % 256);

    if (l <= OUTPUT_SIZE)
    {
      hardware_.write(message_out, l);
      return l;
    }
    else
    {
      logerror("Message from device dropped: message larger than buffer.");
      return -1;
    }
  }

  /********************************************************************
   * Logging
   */

private:
  void log(char byte, const char * msg)
  {
    rosserial_msgs::Log l;
    l.level = byte;
    l.msg = (char*)msg;
    publish(rosserial_msgs::TopicInfo::ID_LOG, &l);
  }

public:
  void logdebug(const char* msg)
  {
    log(rosserial_msgs::Log::ROSDEBUG, msg);
  }
  void loginfo(const char * msg)
  {
    log(rosserial_msgs::Log::INFO, msg);
  }
  void logwarn(const char *msg)
  {
    log(rosserial_msgs::Log::WARN, msg);
  }
  void logerror(const char*msg)
  {
    log(rosserial_msgs::Log::ERROR, msg);
  }
  void logfatal(const char*msg)
  {
    log(rosserial_msgs::Log::FATAL, msg);
  }

  /********************************************************************
   * Parameters
   */

private:
  bool param_recieved;
  rosserial_msgs::RequestParamResponse req_param_resp;

  bool requestParam(const char * name, int time_out =  1000)
  {
    param_recieved = false;
    rosserial_msgs::RequestParamRequest req;
    req.name  = (char*)name;
    publish(TopicInfo::ID_PARAMETER_REQUEST, &req);
    uint32_t end_time = hardware_.time() + time_out;
    while (!param_recieved)
    {
      spinOnce();
      if (hardware_.time() > end_time)
      {
        logwarn("Failed to get param: timeout expired");
        return false;
      }
    }
    return true;
  }

public:
  bool getParam(const char* name, int* param, int length = 1, int timeout = 1000)
  {
    if (requestParam(name, timeout))
    {
      if (length == req_param_resp.ints_length)
      {
        //copy it over
        for (int i = 0; i < length; i++)
          param[i] = req_param_resp.ints[i];
        return true;
      }
      else
      {
        logwarn("Failed to get param: length mismatch");
      }
    }
    return false;
  }
  bool getParam(const char* name, float* param, int length = 1, int timeout = 1000)
  {
    if (requestParam(name, timeout))
    {
      if (length == req_param_resp.floats_length)
      {
        //copy it over
        for (int i = 0; i < length; i++)
          param[i] = req_param_resp.floats[i];
        return true;
      }
      else
      {
        logwarn("Failed to get param: length mismatch");
      }
    }
    return false;
  }
  bool getParam(const char* name, char** param, int length = 1, int timeout = 1000)
  {
    if (requestParam(name, timeout))
    {
      if (length == req_param_resp.strings_length)
      {
        //copy it over
        for (int i = 0; i < length; i++)
          strcpy(param[i], req_param_resp.strings[i]);
        return true;
      }
      else
      {
        logwarn("Failed to get param: length mismatch");
      }
    }
    return false;
  }
  bool getParam(const char* name, bool* param, int length = 1, int timeout = 1000)
  {
    if (requestParam(name, timeout))
    {
      if (length == req_param_resp.ints_length)
      {
        //copy it over
        for (int i = 0; i < length; i++)
          param[i] = req_param_resp.ints[i];
        return true;
      }
      else
      {
        logwarn("Failed to get param: length mismatch");
      }
    }
    return false;
  }
};

}

#endif
```

#### service_client.h
```c
/*
 * Software License Agreement (BSD License)
 *
 * Copyright (c) 2011, Willow Garage, Inc.
 * All rights reserved.
 *
 * Redistribution and use in source and binary forms, with or without
 * modification, are permitted provided that the following conditions
 * are met:
 *
 *  * Redistributions of source code must retain the above copyright
 *    notice, this list of conditions and the following disclaimer.
 *  * Redistributions in binary form must reproduce the above
 *    copyright notice, this list of conditions and the following
 *    disclaimer in the documentation and/or other materials provided
 *    with the distribution.
 *  * Neither the name of Willow Garage, Inc. nor the names of its
 *    contributors may be used to endorse or promote prducts derived
 *    from this software without specific prior written permission.
 *
 * THIS SOFTWARE IS PROVIDED BY THE COPYRIGHT HOLDERS AND CONTRIBUTORS
 * "AS IS" AND ANY EXPRESS OR IMPLIED WARRANTIES, INCLUDING, BUT NOT
 * LIMITED TO, THE IMPLIED WARRANTIES OF MERCHANTABILITY AND FITNESS
 * FOR A PARTICULAR PURPOSE ARE DISCLAIMED. IN NO EVENT SHALL THE
 * COPYRIGHT OWNER OR CONTRIBUTORS BE LIABLE FOR ANY DIRECT, INDIRECT,
 * INCIDENTAL, SPECIAL, EXEMPLARY, OR CONSEQUENTIAL DAMAGES (INCLUDING,
 * BUT NOT LIMITED TO, PROCUREMENT OF SUBSTITUTE GOODS OR SERVICES;
 * LOSS OF USE, DATA, OR PROFITS; OR BUSINESS INTERRUPTION) HOWEVER
 * CAUSED AND ON ANY THEORY OF LIABILITY, WHETHER IN CONTRACT, STRICT
 * LIABILITY, OR TORT (INCLUDING NEGLIGENCE OR OTHERWISE) ARISING IN
 * ANY WAY OUT OF THE USE OF THIS SOFTWARE, EVEN IF ADVISED OF THE
 * POSSIBILITY OF SUCH DAMAGE.
 */

#ifndef _ROS_SERVICE_CLIENT_H_
#define _ROS_SERVICE_CLIENT_H_

#include "../rosserial_msgs/TopicInfo.h"

#include "../ros/publisher.h"
#include "../ros/subscriber.h"

namespace ros
{

template<typename MReq , typename MRes>
class ServiceClient : public Subscriber_
{
public:
  ServiceClient(const char* topic_name) :
    pub(topic_name, &req, rosserial_msgs::TopicInfo::ID_SERVICE_CLIENT + rosserial_msgs::TopicInfo::ID_PUBLISHER)
  {
    this->topic_ = topic_name;
    this->waiting = true;
  }

  virtual void call(const MReq & request, MRes & response)
  {
    if (!pub.nh_->connected()) return;
    ret = &response;
    waiting = true;
    pub.publish(&request);
    while (waiting && pub.nh_->connected())
      if (pub.nh_->spinOnce() < 0) break;
  }

  // these refer to the subscriber
  virtual void callback(unsigned char *data)
  {
    ret->deserialize(data);
    waiting = false;
  }
  virtual const char * getMsgType()
  {
    return this->resp.getType();
  }
  virtual const char * getMsgMD5()
  {
    return this->resp.getMD5();
  }
  virtual int getEndpointType()
  {
    return rosserial_msgs::TopicInfo::ID_SERVICE_CLIENT + rosserial_msgs::TopicInfo::ID_SUBSCRIBER;
  }

  MReq req;
  MRes resp;
  MRes * ret;
  bool waiting;
  Publisher pub;
};

}

#endif
```

#### service_server.h
```c
/*
 * Software License Agreement (BSD License)
 *
 * Copyright (c) 2011, Willow Garage, Inc.
 * All rights reserved.
 *
 * Redistribution and use in source and binary forms, with or without
 * modification, are permitted provided that the following conditions
 * are met:
 *
 *  * Redistributions of source code must retain the above copyright
 *    notice, this list of conditions and the following disclaimer.
 *  * Redistributions in binary form must reproduce the above
 *    copyright notice, this list of conditions and the following
 *    disclaimer in the documentation and/or other materials provided
 *    with the distribution.
 *  * Neither the name of Willow Garage, Inc. nor the names of its
 *    contributors may be used to endorse or promote prducts derived
 *    from this software without specific prior written permission.
 *
 * THIS SOFTWARE IS PROVIDED BY THE COPYRIGHT HOLDERS AND CONTRIBUTORS
 * "AS IS" AND ANY EXPRESS OR IMPLIED WARRANTIES, INCLUDING, BUT NOT
 * LIMITED TO, THE IMPLIED WARRANTIES OF MERCHANTABILITY AND FITNESS
 * FOR A PARTICULAR PURPOSE ARE DISCLAIMED. IN NO EVENT SHALL THE
 * COPYRIGHT OWNER OR CONTRIBUTORS BE LIABLE FOR ANY DIRECT, INDIRECT,
 * INCIDENTAL, SPECIAL, EXEMPLARY, OR CONSEQUENTIAL DAMAGES (INCLUDING,
 * BUT NOT LIMITED TO, PROCUREMENT OF SUBSTITUTE GOODS OR SERVICES;
 * LOSS OF USE, DATA, OR PROFITS; OR BUSINESS INTERRUPTION) HOWEVER
 * CAUSED AND ON ANY THEORY OF LIABILITY, WHETHER IN CONTRACT, STRICT
 * LIABILITY, OR TORT (INCLUDING NEGLIGENCE OR OTHERWISE) ARISING IN
 * ANY WAY OUT OF THE USE OF THIS SOFTWARE, EVEN IF ADVISED OF THE
 * POSSIBILITY OF SUCH DAMAGE.
 */

#ifndef _ROS_SERVICE_SERVER_H_
#define _ROS_SERVICE_SERVER_H_

#include "../rosserial_msgs/TopicInfo.h"

#include "../ros/publisher.h"
#include "../ros/subscriber.h"

namespace ros
{

template<typename MReq , typename MRes, typename ObjT = void>
class ServiceServer : public Subscriber_
{
public:
  typedef void(ObjT::*CallbackT)(const MReq&,  MRes&);

  ServiceServer(const char* topic_name, CallbackT cb, ObjT* obj) :
    pub(topic_name, &resp, rosserial_msgs::TopicInfo::ID_SERVICE_SERVER + rosserial_msgs::TopicInfo::ID_PUBLISHER),
    obj_(obj)
  {
    this->topic_ = topic_name;
    this->cb_ = cb;
  }

  // these refer to the subscriber
  virtual void callback(unsigned char *data)
  {
    req.deserialize(data);
    (obj_->*cb_)(req, resp);
    pub.publish(&resp);
  }
  virtual const char * getMsgType()
  {
    return this->req.getType();
  }
  virtual const char * getMsgMD5()
  {
    return this->req.getMD5();
  }
  virtual int getEndpointType()
  {
    return rosserial_msgs::TopicInfo::ID_SERVICE_SERVER + rosserial_msgs::TopicInfo::ID_SUBSCRIBER;
  }

  MReq req;
  MRes resp;
  Publisher pub;
private:
  CallbackT cb_;
  ObjT* obj_;
};

template<typename MReq , typename MRes>
class ServiceServer<MReq, MRes, void> : public Subscriber_
{
public:
  typedef void(*CallbackT)(const MReq&,  MRes&);

  ServiceServer(const char* topic_name, CallbackT cb) :
    pub(topic_name, &resp, rosserial_msgs::TopicInfo::ID_SERVICE_SERVER + rosserial_msgs::TopicInfo::ID_PUBLISHER)
  {
    this->topic_ = topic_name;
    this->cb_ = cb;
  }

  // these refer to the subscriber
  virtual void callback(unsigned char *data)
  {
    req.deserialize(data);
    cb_(req, resp);
    pub.publish(&resp);
  }
  virtual const char * getMsgType()
  {
    return this->req.getType();
  }
  virtual const char * getMsgMD5()
  {
    return this->req.getMD5();
  }
  virtual int getEndpointType()
  {
    return rosserial_msgs::TopicInfo::ID_SERVICE_SERVER + rosserial_msgs::TopicInfo::ID_SUBSCRIBER;
  }

  MReq req;
  MRes resp;
  Publisher pub;
private:
  CallbackT cb_;
};

}

#endif
```

#### subscriber.h
```c
/*
 * Software License Agreement (BSD License)
 *
 * Copyright (c) 2011, Willow Garage, Inc.
 * All rights reserved.
 *
 * Redistribution and use in source and binary forms, with or without
 * modification, are permitted provided that the following conditions
 * are met:
 *
 *  * Redistributions of source code must retain the above copyright
 *    notice, this list of conditions and the following disclaimer.
 *  * Redistributions in binary form must reproduce the above
 *    copyright notice, this list of conditions and the following
 *    disclaimer in the documentation and/or other materials provided
 *    with the distribution.
 *  * Neither the name of Willow Garage, Inc. nor the names of its
 *    contributors may be used to endorse or promote prducts derived
 *    from this software without specific prior written permission.
 *
 * THIS SOFTWARE IS PROVIDED BY THE COPYRIGHT HOLDERS AND CONTRIBUTORS
 * "AS IS" AND ANY EXPRESS OR IMPLIED WARRANTIES, INCLUDING, BUT NOT
 * LIMITED TO, THE IMPLIED WARRANTIES OF MERCHANTABILITY AND FITNESS
 * FOR A PARTICULAR PURPOSE ARE DISCLAIMED. IN NO EVENT SHALL THE
 * COPYRIGHT OWNER OR CONTRIBUTORS BE LIABLE FOR ANY DIRECT, INDIRECT,
 * INCIDENTAL, SPECIAL, EXEMPLARY, OR CONSEQUENTIAL DAMAGES (INCLUDING,
 * BUT NOT LIMITED TO, PROCUREMENT OF SUBSTITUTE GOODS OR SERVICES;
 * LOSS OF USE, DATA, OR PROFITS; OR BUSINESS INTERRUPTION) HOWEVER
 * CAUSED AND ON ANY THEORY OF LIABILITY, WHETHER IN CONTRACT, STRICT
 * LIABILITY, OR TORT (INCLUDING NEGLIGENCE OR OTHERWISE) ARISING IN
 * ANY WAY OUT OF THE USE OF THIS SOFTWARE, EVEN IF ADVISED OF THE
 * POSSIBILITY OF SUCH DAMAGE.
 */

#ifndef ROS_SUBSCRIBER_H_
#define ROS_SUBSCRIBER_H_

#include "../rosserial_msgs/TopicInfo.h"
#include "../voice_interaction_robot_msgs/FulfilledVoiceCommand.h"

namespace ros
{

/* Base class for objects subscribers. */
class Subscriber_
{
public:
  virtual void callback(unsigned char *data) = 0;
  virtual int getEndpointType() = 0;

  // id_ is set by NodeHandle when we advertise
  int id_;

  virtual const char * getMsgType() = 0;
  virtual const char * getMsgMD5() = 0;
  const char * topic_;
};

/* Bound function subscriber. */
template<typename MsgT, typename ObjT = void>
class Subscriber: public Subscriber_
{
public:
  typedef void(ObjT::*CallbackT)(const MsgT&);
  MsgT msg;

  Subscriber(const char * topic_name, CallbackT cb, ObjT* obj, int endpoint = rosserial_msgs::TopicInfo::ID_SUBSCRIBER) :
    cb_(cb),
    obj_(obj),
    endpoint_(endpoint)
  {
    topic_ = topic_name;
  };

  virtual void callback(unsigned char* data)
  {
    msg.deserialize(data);
    (obj_->*cb_)(msg);
  }

  virtual const char * getMsgType()
  {
    return this->msg.getType();
  }
  virtual const char * getMsgMD5()
  {
    return this->msg.getMD5();
  }
  virtual int getEndpointType()
  {
    return endpoint_;
  }

private:
  CallbackT cb_;
  ObjT* obj_;
  int endpoint_;
};

/* Standalone function subscriber. */
template<typename MsgT>
class Subscriber<MsgT, void>: public Subscriber_
{
public:
  typedef voice_interaction_robot_msgs::FulfilledVoiceCommand(*CallbackT)(const MsgT&);
  MsgT msg;

  Subscriber(const char * topic_name, CallbackT cb, int endpoint = rosserial_msgs::TopicInfo::ID_SUBSCRIBER) :
    cb_(cb),
    endpoint_(endpoint)
  {
    topic_ = topic_name;
	callbackCounter_ = 0;
  };

  virtual void callback(unsigned char* data)
  {
    msg.deserialize(data);
	callbackCounter_ = callbackCounter_ + 1;
    fulfilledCommand_ = this->cb_(msg);
  }

  virtual const char * getMsgType()
  {
    return this->msg.getType();
  }
  virtual const char * getMsgMD5()
  {
    return this->msg.getMD5();
  }
  virtual int getEndpointType()
  {
    return endpoint_;
  }
  voice_interaction_robot_msgs::FulfilledVoiceCommand fulfilledCommand_;
  UDINT callbackCounter_;

private:
  CallbackT cb_;
  int endpoint_;
};

}

#endif
```

#### time.h
```c
/*
 * Software License Agreement (BSD License)
 *
 * Copyright (c) 2011, Willow Garage, Inc.
 * All rights reserved.
 *
 * Redistribution and use in source and binary forms, with or without
 * modification, are permitted provided that the following conditions
 * are met:
 *
 *  * Redistributions of source code must retain the above copyright
 *    notice, this list of conditions and the following disclaimer.
 *  * Redistributions in binary form must reproduce the above
 *    copyright notice, this list of conditions and the following
 *    disclaimer in the documentation and/or other materials provided
 *    with the distribution.
 *  * Neither the name of Willow Garage, Inc. nor the names of its
 *    contributors may be used to endorse or promote prducts derived
 *    from this software without specific prior written permission.
 *
 * THIS SOFTWARE IS PROVIDED BY THE COPYRIGHT HOLDERS AND CONTRIBUTORS
 * "AS IS" AND ANY EXPRESS OR IMPLIED WARRANTIES, INCLUDING, BUT NOT
 * LIMITED TO, THE IMPLIED WARRANTIES OF MERCHANTABILITY AND FITNESS
 * FOR A PARTICULAR PURPOSE ARE DISCLAIMED. IN NO EVENT SHALL THE
 * COPYRIGHT OWNER OR CONTRIBUTORS BE LIABLE FOR ANY DIRECT, INDIRECT,
 * INCIDENTAL, SPECIAL, EXEMPLARY, OR CONSEQUENTIAL DAMAGES (INCLUDING,
 * BUT NOT LIMITED TO, PROCUREMENT OF SUBSTITUTE GOODS OR SERVICES;
 * LOSS OF USE, DATA, OR PROFITS; OR BUSINESS INTERRUPTION) HOWEVER
 * CAUSED AND ON ANY THEORY OF LIABILITY, WHETHER IN CONTRACT, STRICT
 * LIABILITY, OR TORT (INCLUDING NEGLIGENCE OR OTHERWISE) ARISING IN
 * ANY WAY OUT OF THE USE OF THIS SOFTWARE, EVEN IF ADVISED OF THE
 * POSSIBILITY OF SUCH DAMAGE.
 */

#ifndef ROS_TIME_H_
#define ROS_TIME_H_

#include "../ros/duration.h"
#include <math.h>
#include <stdint.h>

namespace ros
{
void normalizeSecNSec(uint32_t &sec, uint32_t &nsec);

class Time
{
public:
  uint32_t sec, nsec;

  Time() : sec(0), nsec(0) {}
  Time(uint32_t _sec, uint32_t _nsec) : sec(_sec), nsec(_nsec)
  {
    normalizeSecNSec(sec, nsec);
  }

  double toSec() const
  {
    return (double)sec + 1e-9 * (double)nsec;
  };
  void fromSec(double t)
  {
    sec = (uint32_t) floor(t);
    nsec = (uint32_t) round((t - sec) * 1e9);
  };

  uint32_t toNsec()
  {
    return (uint32_t)sec * 1000000000ull + (uint32_t)nsec;
  };
  Time& fromNSec(int32_t t);

  Time& operator +=(const Duration &rhs);
  Time& operator -=(const Duration &rhs);

  static Time now();
  static void setNow(Time & new_now);
};

}

#endif
```

#### Twist.h
```c
#ifndef _ROS_geometry_msgs_Twist_h
#define _ROS_geometry_msgs_Twist_h

#include <stdint.h>
#include <string.h>
#include <stdlib.h>
#include "../../RosNode/ros/msg.h"
#include "../geometry_msgs/Vector3.h"

namespace geometry_msgs
{

  class Twist : public ros::Msg
  {
    public:
      typedef geometry_msgs::Vector3 _linear_type;
      _linear_type linear;
      typedef geometry_msgs::Vector3 _angular_type;
      _angular_type angular;

    Twist():
      linear(),
      angular()
    {
    }

    virtual int serialize(unsigned char *outbuffer) const
    {
      int offset = 0;
      offset += this->linear.serialize(outbuffer + offset);
      offset += this->angular.serialize(outbuffer + offset);
      return offset;
    }

    virtual int deserialize(unsigned char *inbuffer)
    {
      int offset = 0;
      offset += this->linear.deserialize(inbuffer + offset);
      offset += this->angular.deserialize(inbuffer + offset);
     return offset;
    }

    const char * getType(){ return "geometry_msgs/Twist"; };
    const char * getMD5(){ return "9f195f881246fdfa2798d1d3eebca84a"; };

  };

}
#endif
```

#### Vector3.h
```c
#ifndef _ROS_geometry_msgs_Vector3_h
#define _ROS_geometry_msgs_Vector3_h

#include <stdint.h>
#include <string.h>
#include <stdlib.h>
#include "../../RosNode/ros/msg.h"

namespace geometry_msgs
{

  class Vector3 : public ros::Msg
  {
    public:
      typedef float _x_type;
      _x_type x;
      typedef float _y_type;
      _y_type y;
      typedef float _z_type;
      _z_type z;

    Vector3():
      x(0),
      y(0),
      z(0)
    {
    }

    virtual int serialize(unsigned char *outbuffer) const
    {
      int offset = 0;
      offset += serializeAvrFloat64(outbuffer + offset, this->x);
      offset += serializeAvrFloat64(outbuffer + offset, this->y);
      offset += serializeAvrFloat64(outbuffer + offset, this->z);
      return offset;
    }

    virtual int deserialize(unsigned char *inbuffer)
    {
      int offset = 0;
      offset += deserializeAvrFloat64(inbuffer + offset, &(this->x));
      offset += deserializeAvrFloat64(inbuffer + offset, &(this->y));
      offset += deserializeAvrFloat64(inbuffer + offset, &(this->z));
     return offset;
    }

    const char * getType(){ return "geometry_msgs/Vector3"; };
    const char * getMD5(){ return "4a842b65f413084dc2b10fb484ea7f17"; };

  };

}
#endif
```

#### Log.h
```c
#ifndef _ROS_rosserial_msgs_Log_h
#define _ROS_rosserial_msgs_Log_h

#include <stdint.h>
#include <string.h>
#include <stdlib.h>
#include "../ros/msg.h"

namespace rosserial_msgs
{

  class Log : public ros::Msg
  {
    public:
      typedef uint8_t _level_type;
      _level_type level;
      typedef const char* _msg_type;
      _msg_type msg;
      enum { ROSDEBUG = 0 };
      enum { INFO = 1 };
      enum { WARN = 2 };
      enum { ERROR = 3 };
      enum { FATAL = 4 };

    Log():
      level(0),
      msg("")
    {
    }

    virtual int serialize(unsigned char *outbuffer) const
    {
      int offset = 0;
      *(outbuffer + offset + 0) = (this->level >> (8 * 0)) & 0xFF;
      offset += sizeof(this->level);
      uint32_t length_msg = strlen(this->msg);
      varToArr(outbuffer + offset, length_msg);
      offset += 4;
      memcpy(outbuffer + offset, this->msg, length_msg);
      offset += length_msg;
      return offset;
    }

    virtual int deserialize(unsigned char *inbuffer)
    {
      int offset = 0;
      this->level =  ((uint8_t) (*(inbuffer + offset)));
      offset += sizeof(this->level);
      uint32_t length_msg;
      arrToVar(length_msg, (inbuffer + offset));
      offset += 4;
      for(unsigned int k= offset; k< offset+length_msg; ++k){
          inbuffer[k-1]=inbuffer[k];
      }
      inbuffer[offset+length_msg-1]=0;
      this->msg = (char *)(inbuffer + offset-1);
      offset += length_msg;
     return offset;
    }

    const char * getType(){ return "rosserial_msgs/Log"; };
    const char * getMD5(){ return "11abd731c25933261cd6183bd12d6295"; };

  };

}
#endif
```

#### TopicInfo.h
```c
#ifndef _ROS_rosserial_msgs_TopicInfo_h
#define _ROS_rosserial_msgs_TopicInfo_h

#include <stdint.h>
#include <string.h>
#include <stdlib.h>
#include "../ros/msg.h"

namespace rosserial_msgs
{

  class TopicInfo : public ros::Msg
  {
    public:
      typedef uint16_t _topic_id_type;
      _topic_id_type topic_id;
      typedef const char* _topic_name_type;
      _topic_name_type topic_name;
      typedef const char* _message_type_type;
      _message_type_type message_type;
      typedef const char* _md5sum_type;
      _md5sum_type md5sum;
      typedef int32_t _buffer_size_type;
      _buffer_size_type buffer_size;
      enum { ID_PUBLISHER = 0 };
      enum { ID_SUBSCRIBER = 1 };
      enum { ID_SERVICE_SERVER = 2 };
      enum { ID_SERVICE_CLIENT = 4 };
      enum { ID_PARAMETER_REQUEST = 6 };
      enum { ID_LOG = 7 };
      enum { ID_TIME = 10 };
      enum { ID_TX_STOP = 11 };

    TopicInfo():
      topic_id(0),
      topic_name(""),
      message_type(""),
      md5sum(""),
      buffer_size(0)
    {
    }

    virtual int serialize(unsigned char *outbuffer) const
    {
      int offset = 0;
      *(outbuffer + offset + 0) = (this->topic_id >> (8 * 0)) & 0xFF;
      *(outbuffer + offset + 1) = (this->topic_id >> (8 * 1)) & 0xFF;
      offset += sizeof(this->topic_id);
      uint32_t length_topic_name = strlen(this->topic_name);
      varToArr(outbuffer + offset, length_topic_name);
      offset += 4;
      memcpy(outbuffer + offset, this->topic_name, length_topic_name);
      offset += length_topic_name;
      uint32_t length_message_type = strlen(this->message_type);
      varToArr(outbuffer + offset, length_message_type);
      offset += 4;
      memcpy(outbuffer + offset, this->message_type, length_message_type);
      offset += length_message_type;
      uint32_t length_md5sum = strlen(this->md5sum);
      varToArr(outbuffer + offset, length_md5sum);
      offset += 4;
      memcpy(outbuffer + offset, this->md5sum, length_md5sum);
      offset += length_md5sum;
      union {
        int32_t real;
        uint32_t base;
      } u_buffer_size;
      u_buffer_size.real = this->buffer_size;
      *(outbuffer + offset + 0) = (u_buffer_size.base >> (8 * 0)) & 0xFF;
      *(outbuffer + offset + 1) = (u_buffer_size.base >> (8 * 1)) & 0xFF;
      *(outbuffer + offset + 2) = (u_buffer_size.base >> (8 * 2)) & 0xFF;
      *(outbuffer + offset + 3) = (u_buffer_size.base >> (8 * 3)) & 0xFF;
      offset += sizeof(this->buffer_size);
      return offset;
    }

    virtual int deserialize(unsigned char *inbuffer)
    {
      int offset = 0;
      this->topic_id =  ((uint16_t) (*(inbuffer + offset)));
      this->topic_id |= ((uint16_t) (*(inbuffer + offset + 1))) << (8 * 1);
      offset += sizeof(this->topic_id);
      uint32_t length_topic_name;
      arrToVar(length_topic_name, (inbuffer + offset));
      offset += 4;
      for(unsigned int k= offset; k< offset+length_topic_name; ++k){
          inbuffer[k-1]=inbuffer[k];
      }
      inbuffer[offset+length_topic_name-1]=0;
      this->topic_name = (char *)(inbuffer + offset-1);
      offset += length_topic_name;
      uint32_t length_message_type;
      arrToVar(length_message_type, (inbuffer + offset));
      offset += 4;
      for(unsigned int k= offset; k< offset+length_message_type; ++k){
          inbuffer[k-1]=inbuffer[k];
      }
      inbuffer[offset+length_message_type-1]=0;
      this->message_type = (char *)(inbuffer + offset-1);
      offset += length_message_type;
      uint32_t length_md5sum;
      arrToVar(length_md5sum, (inbuffer + offset));
      offset += 4;
      for(unsigned int k= offset; k< offset+length_md5sum; ++k){
          inbuffer[k-1]=inbuffer[k];
      }
      inbuffer[offset+length_md5sum-1]=0;
      this->md5sum = (char *)(inbuffer + offset-1);
      offset += length_md5sum;
      union {
        int32_t real;
        uint32_t base;
      } u_buffer_size;
      u_buffer_size.base = 0;
      u_buffer_size.base |= ((uint32_t) (*(inbuffer + offset + 0))) << (8 * 0);
      u_buffer_size.base |= ((uint32_t) (*(inbuffer + offset + 1))) << (8 * 1);
      u_buffer_size.base |= ((uint32_t) (*(inbuffer + offset + 2))) << (8 * 2);
      u_buffer_size.base |= ((uint32_t) (*(inbuffer + offset + 3))) << (8 * 3);
      this->buffer_size = u_buffer_size.real;
      offset += sizeof(this->buffer_size);
     return offset;
    }

    const char * getType(){ return "rosserial_msgs/TopicInfo"; };
    const char * getMD5(){ return "0ad51f88fc44892f8c10684077646005"; };

  };

}
#endif
```

#### SoundRequest.h
```c
#ifndef _ROS_sound_play_SoundRequest_h
#define _ROS_sound_play_SoundRequest_h

#include <stdint.h>
#include <string.h>
#include <stdlib.h>
#include "../ros/msg.h"

namespace sound_play
{

  class SoundRequest : public ros::Msg
  {
    public:
      typedef int8_t _sound_type;
      _sound_type sound;
      typedef int8_t _command_type;
      _command_type command;
      typedef float _volume_type;
      _volume_type volume;
      typedef const char* _arg_type;
      _arg_type arg;
      typedef const char* _arg2_type;
      _arg2_type arg2;
      enum { BACKINGUP =  1 };
      enum { NEEDS_UNPLUGGING =  2 };
      enum { NEEDS_PLUGGING =  3 };
      enum { NEEDS_UNPLUGGING_BADLY =  4 };
      enum { NEEDS_PLUGGING_BADLY =  5 };
      enum { ALL =  -1  };
      enum { PLAY_FILE =  -2 };
      enum { SAY =  -3 };
      enum { PLAY_STOP =  0  };
      enum { PLAY_ONCE =  1  };
      enum { PLAY_START =  2  };

    SoundRequest():
      sound(0),
      command(0),
      volume(0),
      arg(""),
      arg2("")
    {
    }

    virtual int serialize(unsigned char *outbuffer) const
    {
      int offset = 0;
      union {
        int8_t real;
        uint8_t base;
      } u_sound;
      u_sound.real = this->sound;
      *(outbuffer + offset + 0) = (u_sound.base >> (8 * 0)) & 0xFF;
      offset += sizeof(this->sound);
      union {
        int8_t real;
        uint8_t base;
      } u_command;
      u_command.real = this->command;
      *(outbuffer + offset + 0) = (u_command.base >> (8 * 0)) & 0xFF;
      offset += sizeof(this->command);
      union {
        float real;
        uint32_t base;
      } u_volume;
      u_volume.real = this->volume;
      *(outbuffer + offset + 0) = (u_volume.base >> (8 * 0)) & 0xFF;
      *(outbuffer + offset + 1) = (u_volume.base >> (8 * 1)) & 0xFF;
      *(outbuffer + offset + 2) = (u_volume.base >> (8 * 2)) & 0xFF;
      *(outbuffer + offset + 3) = (u_volume.base >> (8 * 3)) & 0xFF;
      offset += sizeof(this->volume);
      uint32_t length_arg = strlen(this->arg);
      varToArr(outbuffer + offset, length_arg);
      offset += 4;
      memcpy(outbuffer + offset, this->arg, length_arg);
      offset += length_arg;
      uint32_t length_arg2 = strlen(this->arg2);
      varToArr(outbuffer + offset, length_arg2);
      offset += 4;
      memcpy(outbuffer + offset, this->arg2, length_arg2);
      offset += length_arg2;
      return offset;
    }

    virtual int deserialize(unsigned char *inbuffer)
    {
      int offset = 0;
      union {
        int8_t real;
        uint8_t base;
      } u_sound;
      u_sound.base = 0;
      u_sound.base |= ((uint8_t) (*(inbuffer + offset + 0))) << (8 * 0);
      this->sound = u_sound.real;
      offset += sizeof(this->sound);
      union {
        int8_t real;
        uint8_t base;
      } u_command;
      u_command.base = 0;
      u_command.base |= ((uint8_t) (*(inbuffer + offset + 0))) << (8 * 0);
      this->command = u_command.real;
      offset += sizeof(this->command);
      union {
        float real;
        uint32_t base;
      } u_volume;
      u_volume.base = 0;
      u_volume.base |= ((uint32_t) (*(inbuffer + offset + 0))) << (8 * 0);
      u_volume.base |= ((uint32_t) (*(inbuffer + offset + 1))) << (8 * 1);
      u_volume.base |= ((uint32_t) (*(inbuffer + offset + 2))) << (8 * 2);
      u_volume.base |= ((uint32_t) (*(inbuffer + offset + 3))) << (8 * 3);
      this->volume = u_volume.real;
      offset += sizeof(this->volume);
      uint32_t length_arg;
      arrToVar(length_arg, (inbuffer + offset));
      offset += 4;
      for(unsigned int k= offset; k< offset+length_arg; ++k){
          inbuffer[k-1]=inbuffer[k];
      }
      inbuffer[offset+length_arg-1]=0;
      this->arg = (char *)(inbuffer + offset-1);
      offset += length_arg;
      uint32_t length_arg2;
      arrToVar(length_arg2, (inbuffer + offset));
      offset += 4;
      for(unsigned int k= offset; k< offset+length_arg2; ++k){
          inbuffer[k-1]=inbuffer[k];
      }
      inbuffer[offset+length_arg2-1]=0;
      this->arg2 = (char *)(inbuffer + offset-1);
      offset += length_arg2;
     return offset;
    }

    const char * getType(){ return "sound_play/SoundRequest"; };
    const char * getMD5(){ return "d098ce4a040686259137ece23a625167"; };

  };

}
#endif
```

### Library Logical/Libraries/RosWrap (ANSIC)

#### Types.typ - Exported data types
```iecst
TYPE
	RosWrapper_Internal_Type : 	STRUCT
		Ident : UDINT;
		OldWakeCommand : BOOL;
	END_STRUCT;
	RosWrapper_Velocity_Type : 	STRUCT
		linear : Vector3_Type;
		angular : Vector3_Type;
	END_STRUCT;
	Vector3_Type : 	STRUCT
		x : REAL;
		y : REAL;
		z : REAL;
	END_STRUCT;
	RosWrapper_Slot_Type : 	STRUCT
		Key : STRING[80];
		Value : STRING[80];
	END_STRUCT;
	RosWrapper_FulfilledCommand_Type : 	STRUCT
		IntentName : STRING[80];
		NumSlots : UDINT;
		Slot : ARRAY[0..ROS_MAX_SLOT_INDEX]OF RosWrapper_Slot_Type;
	END_STRUCT;
END_TYPE
```

#### Constants.var - Exported constants
```iecst
VAR CONSTANT
	ROS_MAX_SLOT_INDEX : UDINT := 9;
END_VAR
```

#### RosWrap.fun - Exported functions and function blocks
```iecst
{REDUND_ERROR} FUNCTION_BLOCK RosWrapper (*TODO: Add your comment here*) (*$GROUP=User,$CAT=User,$GROUPICON=User.png,$CATICON=User.png*)
	VAR_INPUT
		Enable : {REDUND_UNREPLICABLE} BOOL;
		WakeCommand : BOOL;
	END_VAR
	VAR_OUTPUT
		Active : BOOL;
		Error : BOOL;
		ErrorID : UINT;
		FulfilledCommand : RosWrapper_FulfilledCommand_Type;
	END_VAR
	VAR
		Internal : RosWrapper_Internal_Type;
	END_VAR
END_FUNCTION_BLOCK
```

#### RosWrapper.cpp
```cpp
#include <bur/plctypes.h>
#include "RosWrap.h"
#include "../RosNode/rosnode.hpp"

// amount of memory to be allocated for heap storage must be specified for every ANSI C++ program with the bur_heap_size variable
unsigned long bur_heap_size = 0xFFFF;

void RosWrapper(struct RosWrapper* Inst)
{
	static std_msgs::String wakeWord;
	static BOOL wakeCommand;

	static voice_interaction_robot_msgs::FulfilledVoiceCommand fulfilledCommand;

	if (Inst == 0)
		return;

	if (Inst->Enable == true)
	{
		// The first time the FB gets here after being enabled, setup operations are carried out
		if (Inst->Internal.Ident == 0)
		{
			// Constructing the RosNode object based on the input configuration info
			RosNode* NodeInstance = new RosNode();
			Inst->Internal.Ident = reinterpret_cast<UDINT>(NodeInstance);
		}
		else
		{
			// Dereferencing the axis object
			RosNode* NodeInstance = static_cast<RosNode*>((void*)Inst->Internal.Ident);

//			// Mapping parameters from outside world.
//			if ((Inst->WakeCommand) && (!Inst->Internal.OldWakeCommand))
//			{
//				wakeCommand = true;
//				wakeWord.data = "wake";
//			}
//			else
//			{
//				wakeCommand = false;
//				wakeWord.data = "";
//			}

			// Calling the cyclic processing method.
			fulfilledCommand = NodeInstance->Cyclic(wakeWord,wakeCommand);
//			NodeInstance->Cyclic();

			// Post-processing logic to convert the data from any topic subscriptions to useable IEC structures.
			brsmemset((UDINT)&Inst->FulfilledCommand,0,sizeof(Inst->FulfilledCommand));
			if (fulfilledCommand.intent_name != 0)
			{
				// Extracting the intent name
				const char* intent_name = fulfilledCommand.intent_name;
				brsstrcpy((UDINT)Inst->FulfilledCommand.IntentName,(UDINT)intent_name);
				// Extracting the number of slots
				Inst->FulfilledCommand.NumSlots = (UDINT)fulfilledCommand.slots_length;
				// Now extracting data for each individual slot
				for (UINT i = 0; i < ROS_MAX_SLOT_INDEX; i++)
				{
					if (i < fulfilledCommand.slots_length)
					{
						const char* slot_key = fulfilledCommand.slots[i].key;
						brsstrcpy((UDINT)Inst->FulfilledCommand.Slot[i].Key,(UDINT)slot_key);
						const char* slot_value = fulfilledCommand.slots[i].value;
						brsstrcpy((UDINT)Inst->FulfilledCommand.Slot[i].Value,(UDINT)slot_value);
					}
				}
			}
//
//			// Storing old values for edge detection
//			Inst->Internal.OldWakeCommand = Inst->WakeCommand;
		}
	}
}
```

- Visualisation Logical/mappView (not shown)

### Package Logical/MotionObjects - gConveyorobj

### Data object Logical/MotionObjects/gConveyora (Apt)

#### gConveyora.apt
```
AcoposParameterTable:
  Root Parameters:
    110 = ncSW_ON (Name=CMD_SIMULATION)
```

- Data object Logical/MotionObjects/gConveyori (Ax) (no source held here)

### Data object Logical/MotionObjects/acp10etxen (Ett)

- acp10etxen.ett (not shown)

### Program Logical/Programs/main (IEC)

#### Main.st - Init, cyclic, exit code
```iecst
PROGRAM _INIT

	Conveyor.MpLink := ADR(gMpLinkConveyor);
	Conveyor.Axis := ADR(gConveyor);
	Conveyor.Enable := TRUE;
	Conveyor.Parameters := ADR(ConveyorParameters);

	ConveyorParameters.Acceleration := 1;
	ConveyorParameters.Deceleration := 1;
	ConveyorParameters.Jog.Acceleration := ConveyorParameters.Acceleration;
	ConveyorParameters.Jog.Deceleration := ConveyorParameters.Deceleration;
	ConveyorParameters.Jog.Velocity := 1;
	ConveyorParameters.Velocity := 1;

	TON_ShowBox1.PT := T#1.75s;
	TON_ShowBox2.PT := T#1.75s;
	TON_ShowBox3.PT := T#1.75s;

END_PROGRAM

PROGRAM _CYCLIC

	// Scaling from axis units to HMI: 100 pixels = 1 meter.
	// On our SVG, the outer belt has a diameter of 80 pixels. This means that one rev of the belt => 251.3 pixels => 2.513 meters

	ProcessROSCommands;

	// Initializing our axis
	IF (Conveyor.Active) THEN
		Conveyor.Power := TRUE;
		IF (Conveyor.PowerOn) THEN
			Conveyor.Home := TRUE;
		END_IF
		IF (Conveyor.IsHomed) THEN
			Conveyor.Home := FALSE;
		END_IF
	END_IF
	IF (Conveyor.Info.MoveDone) THEN
		Conveyor.MoveAbsolute := FALSE;
		Conveyor.MoveAdditive := FALSE;
	END_IF

	// Detect parameter changes and update on the fly
	IF (((ConveyorParameters.Velocity <> OldParameters.Velocity) OR (ConveyorParameters.Acceleration <> OldParameters.Acceleration) OR
		(ConveyorParameters.Deceleration <> OldParameters.Deceleration)) AND (Conveyor.MoveActive)) THEN
		Conveyor.Update := TRUE;
	END_IF
	IF (Conveyor.UpdateDone) THEN
		Conveyor.Update := FALSE;
	END_IF
	OldParameters := ConveyorParameters;

	CASE AutoStep OF
		STEP_IDLE:
			IF (StartAutoMode) THEN
				ShowBox1 := TRUE;
				NextBoxIndex := 1;
				Conveyor.MoveVelocity := TRUE;
				AutoStep := STEP_AUTO;
			END_IF

		STEP_AUTO:
			IF (NOT StartAutoMode) THEN
				Conveyor.MoveVelocity := FALSE;
				AutoStep := STEP_IDLE;
			ELSIF (NextBoxPosition > 3) THEN
				IF (NextBoxIndex = 1) THEN
					ShowBox2 := TRUE;
				ELSIF (NextBoxIndex = 2) THEN
					ShowBox3 := TRUE;
				ELSIF (NextBoxIndex = 3) THEN
					ShowBox1 := TRUE;
				END_IF
				NextBoxIndex := NextBoxIndex + 1;
			END_IF

	END_CASE

	IF (NextBoxIndex = 1) THEN
		NextBoxPosition := BoxPosition1;
	ELSIF (NextBoxIndex = 2) THEN
		NextBoxPosition := BoxPosition2;
	ELSIF (NextBoxIndex = 3) THEN
		NextBoxPosition := BoxPosition3;
	END_IF

	// Handling the motion of the motors
	IF (Conveyor.IsHomed) THEN
		// Logic to figure out where the motors are
		//	MotorPosition := (360 * fmod(LREAL_TO_REAL(Conveyor.Position),MOTOR_PERIOD) / MOTOR_PERIOD);
		MotorPosition := (360 * LREAL_TO_REAL(Conveyor.Position) / MOTOR_PERIOD);
		brsftoa(MotorPosition,ADR(PositionString));
		Motor1Transform := '{"select":"#motorAxis1","duration":2,"spin":[';
		brsstrcat(ADR(Motor1Transform),ADR(PositionString));
		brsstrcat(ADR(Motor1Transform),ADR(',0,0]}'));
		Motor2Transform := '{"select":"#motorAxis2","duration":2,"spin":[';
		brsstrcat(ADR(Motor2Transform),ADR(PositionString));
		brsstrcat(ADR(Motor2Transform),ADR(',0,0]}'));
		Motor3Transform := '{"select":"#motorAxis3","duration":2,"spin":[';
		brsstrcat(ADR(Motor3Transform),ADR(PositionString));
		brsstrcat(ADR(Motor3Transform),ADR(',0,0]}'));
		Motor4Transform := '{"select":"#motorAxis4","duration":2,"spin":[';
		brsstrcat(ADR(Motor4Transform),ADR(PositionString));
		brsstrcat(ADR(Motor4Transform),ADR(',0,0]}'));
	ELSE
		Motor1Transform := '{"select":"#motorAxis1","duration":2,"spin":[0,0,0]}';
		Motor2Transform := '{"select":"#motorAxis2","duration":2,"spin":[0,0,0]}';
		Motor3Transform := '{"select":"#motorAxis3","duration":2,"spin":[0,0,0]}';
		Motor4Transform := '{"select":"#motorAxis4","duration":2,"spin":[0,0,0]}';
	END_IF

	// Handling the motion of the boxes
	IF (EDGEPOS(ShowBox1)) THEN
		TON_ShowBox1.IN := TRUE;
	END_IF
	IF (TON_ShowBox1.Q) THEN
		TON_ShowBox1.IN := FALSE;
		BoxOffset1 := Conveyor.Position;
	END_IF
	IF (TON_ShowBox1.IN) THEN
		Box1Transform := '{"select":"#box_blue_1","display":true,"duration":1500,"scale":[1.2,1.2],"translate":[0,0]}';
	ELSIF (ShowBox1) THEN
		BoxPosition1 := LREAL_TO_REAL(Conveyor.Position - BoxOffset1);
		Box1Transform := '{"select":"#box_blue_1","display":true,"duration":2,"scale":[1,1],"translate":[';
		brsftoa(LREAL_TO_REAL(BoxPosition1*100),ADR(PositionString));
		brsstrcat(ADR(Box1Transform),ADR(PositionString));
		brsstrcat(ADR(Box1Transform),ADR(',0]}'));
	ELSE
		BoxPosition1 := 0;
		Box1Transform := Box2Transform := '{"select":"#box_blue_1","display":false,"duration":2,"scale":[0.1,0.1],"translate":[40,0]}';
	END_IF
	IF (BoxPosition1 > EXIT_POSITION) THEN
		ShowBox1 := FALSE;
		blueCaseComplete := TRUE;
	END_IF

	IF (EDGEPOS(ShowBox2)) THEN
		TON_ShowBox2.IN := TRUE;
	END_IF
	IF (TON_ShowBox2.Q) THEN
		TON_ShowBox2.IN := FALSE;
		BoxOffset2 := Conveyor.Position;
	END_IF
	IF (TON_ShowBox2.IN) THEN
		Box2Transform := '{"select":"#box_green_2","display":true,"duration":1500,"scale":[1.2,1.2],"translate":[0,0]}';
	ELSIF (ShowBox2) THEN
		BoxPosition2 := LREAL_TO_REAL(Conveyor.Position - BoxOffset2);
		Box2Transform := '{"select":"#box_green_2","display":true,"duration":2,"scale":[1,1],"translate":[';
		brsftoa(LREAL_TO_REAL(BoxPosition2*100),ADR(PositionString));
		brsstrcat(ADR(Box2Transform),ADR(PositionString));
		brsstrcat(ADR(Box2Transform),ADR(',0]}'));
	ELSE
		BoxPosition2 := 0;
		Box2Transform := '{"select":"#box_green_2","display":false,"duration":2,"scale":[0.1,0.1],"translate":[30,0]}';
	END_IF

	IF (BoxPosition2 > EXIT_POSITION) THEN
		ShowBox2 := FALSE;
		greenCaseComplete := TRUE;
	END_IF

	IF (EDGEPOS(ShowBox3)) THEN
		TON_ShowBox3.IN := TRUE;
	END_IF
	IF (TON_ShowBox3.Q) THEN
		TON_ShowBox3.IN := FALSE;
		BoxOffset3 := Conveyor.Position;
	END_IF
	IF (TON_ShowBox3.IN) THEN
		Box3Transform := '{"select":"#box_red_3","display":true,"duration":1500,"scale":[1.2,1.2],"translate":[0,0]}';
	ELSIF (ShowBox3) THEN
		BoxPosition3 := LREAL_TO_REAL(Conveyor.Position - BoxOffset3);
		Box3Transform := '{"select":"#box_red_3","display":true,"duration":2,"scale":[1,1],"translate":[';
		brsftoa(LREAL_TO_REAL(BoxPosition3*100),ADR(PositionString));
		brsstrcat(ADR(Box3Transform),ADR(PositionString));
		brsstrcat(ADR(Box3Transform),ADR(',0]}'));
	ELSE
		BoxPosition3 := 0;
		Box3Transform := '{"select":"#box_red_3","display":false,"duration":2,"scale":[0.1,0.1],"translate":[30,0]}';
	END_IF
	IF (BoxPosition3 > EXIT_POSITION) THEN
		ShowBox3 := FALSE;
		redCaseComplete := TRUE;
	END_IF

	// Handling the light
	IF (WorklightOn) THEN
		WorklightTransform := '{"select":"#work_light_beam","display":true,"duration":2,"translate":[0,0]}';
	ELSE
		WorklightTransform := '{"select":"#work_light_beam","display":false,"duration":2,"translate":[0,0]}';
	END_IF

	// Creating the transform string from all elements
	TotalTransform := '[';
	brsstrcat(ADR(TotalTransform),ADR(WorklightTransform));
	brsstrcat(ADR(TotalTransform),ADR(','));
	brsstrcat(ADR(TotalTransform),ADR(Box1Transform));
	brsstrcat(ADR(TotalTransform),ADR(','));
	brsstrcat(ADR(TotalTransform),ADR(Box2Transform));
	brsstrcat(ADR(TotalTransform),ADR(','));
	brsstrcat(ADR(TotalTransform),ADR(Box3Transform));
	brsstrcat(ADR(TotalTransform),ADR(','));
	brsstrcat(ADR(TotalTransform),ADR(Motor1Transform));
	brsstrcat(ADR(TotalTransform),ADR(','));
	brsstrcat(ADR(TotalTransform),ADR(Motor2Transform));
	brsstrcat(ADR(TotalTransform),ADR(','));
	brsstrcat(ADR(TotalTransform),ADR(Motor3Transform));
	brsstrcat(ADR(TotalTransform),ADR(','));
	brsstrcat(ADR(TotalTransform),ADR(Motor4Transform));
	brsstrcat(ADR(TotalTransform),ADR(']'));

	// Calling the FBs
	Conveyor();
	TON_ShowBox1();
	TON_ShowBox2();
	TON_ShowBox3();

END_PROGRAM

PROGRAM _EXIT
	(* Insert code here *)

END_PROGRAM
```

#### Types.typ - Local data types
```iecst
TYPE
	AutoSteps_enum :
		(
		STEP_IDLE,
		STEP_AUTO
		);
END_TYPE
```

#### Variables.var - Local variables
```iecst
VAR
	NextBoxPosition : REAL;
	AutoStep : AutoSteps_enum;
	StartAutoMode : BOOL;
	NextBoxIndex : USINT;
	TON_ShowBox1 : TON;
	TON_ShowBox2 : TON;
	TON_ShowBox3 : TON;
END_VAR
VAR CONSTANT
	EXIT_POSITION : REAL := 8.5;
END_VAR
VAR
	NotifyBox1 : BOOL;
	NotifyBox2 : BOOL;
	NotifyBox3 : BOOL;
END_VAR
VAR CONSTANT
	NOTIFY_POSITION : REAL := 2;
END_VAR
VAR
	TempString : STRING[80];
	BoxPosition1 : REAL;
	BoxPosition2 : REAL;
	BoxPosition3 : REAL;
	WorklightOn : BOOL;
	ShowBox2 : BOOL;
	ShowBox3 : BOOL;
	BoxOffset2 : LREAL;
	BoxOffset3 : LREAL;
	BoxOffset1 : LREAL;
	ShowBox1 : BOOL;
	MotorPosition : REAL;
END_VAR
VAR CONSTANT
	MOTOR_PERIOD : REAL := 2.513;
END_VAR
VAR
	WorklightTransform : STRING[1000];
	Box1Transform : STRING[1000];
	Box2Transform : STRING[1000];
	Box3Transform : STRING[1000];
	Motor1Transform : STRING[1000];
	Motor2Transform : STRING[1000];
	Motor3Transform : STRING[1000];
	Motor4Transform : STRING[1000];
	TotalTransform : STRING[10000];
	PositionString : STRING[80];
	OldParameters : MpAxisBasicParType;
	ConveyorParameters : MpAxisBasicParType;
	Conveyor : MpAxisBasic;
	LocalCommand : RosWrapper_FulfilledCommand_Type;
	RosWrapper_0 : RosWrapper;
END_VAR
```

#### Action.st
```iecst
ACTION ProcessROSCommands:

	// Command to turn the work light on or off
	IF (ROSCommand.IntentName = 'workLightCommand') THEN
		IF (ROSCommand.Slot[0].Value = 'off') THEN
			WorklightOn := FALSE;
		ELSIF (ROSCommand.Slot[0].Value = 'on') THEN
			WorklightOn := TRUE;
		END_IF
	END_IF

	// Command to jog the axis
	IF (ROSCommand.IntentName = 'jogMove') THEN
		IF (ROSCommand.Slot[0].Value = 'forward') THEN
			ConveyorParameters.Direction := mpAXIS_DIR_POSITIVE;
		ELSIF (ROSCommand.Slot[0].Value = 'backward') THEN
			ConveyorParameters.Direction := mpAXIS_DIR_NEGATIVE;
		END_IF
		ConveyorParameters.Velocity := brsatof(ADR(ROSCommand.Slot[1].Value));
		Conveyor.MoveVelocity := TRUE;
	END_IF

	// Command to move a fixed distance
	IF (ROSCommand.IntentName = 'distanceMove') THEN
		IF (ROSCommand.Slot[0].Value = 'forward') THEN
			ConveyorParameters.Direction := mpAXIS_DIR_POSITIVE;
			ConveyorParameters.Distance := 1 * brsatof(ADR(ROSCommand.Slot[1].Value));
		ELSIF (ROSCommand.Slot[0].Value = 'backward') THEN
			ConveyorParameters.Distance := (-1) * brsatof(ADR(ROSCommand.Slot[1].Value));
			ConveyorParameters.Direction := mpAXIS_DIR_NEGATIVE;
		END_IF
		Conveyor.MoveAdditive := TRUE;
	END_IF

	// Stop command--halts all motion
	IF (ROSCommand.IntentName = 'stop') THEN
		Conveyor.MoveVelocity := FALSE;
		Conveyor.MoveAbsolute := FALSE;
		Conveyor.MoveAdditive := FALSE;
		StartAutoMode := FALSE;
	END_IF

	// Command to change parameter values
	IF (ROSCommand.IntentName = 'setParameter') THEN
		IF (ROSCommand.Slot[0].Value = 'speed') THEN
			ConveyorParameters.Velocity := brsatof(ADR(ROSCommand.Slot[1].Value));
		ELSIF (ROSCommand.Slot[0].Value = 'acceleration') THEN
			ConveyorParameters.Acceleration := brsatof(ADR(ROSCommand.Slot[1].Value));
		ELSIF (ROSCommand.Slot[0].Value = 'deceleration') THEN
			ConveyorParameters.Deceleration := brsatof(ADR(ROSCommand.Slot[1].Value));
		END_IF
	END_IF

	// Case commands: place a case
	IF (ROSCommand.IntentName = 'placeCase') THEN
		IF (ROSCommand.Slot[0].Value = 'Blue') THEN
			ShowBox1 := TRUE;
		ELSIF (ROSCommand.Slot[0].Value = 'Green') THEN
			ShowBox2 := TRUE;
		ELSIF (ROSCommand.Slot[0].Value = 'red') THEN
			ShowBox3 := TRUE;
		END_IF
	END_IF
	// Case commands: clear all cases
	IF (ROSCommand.IntentName = 'clearAllCases') THEN
		ShowBox1 := FALSE;
		ShowBox2 := FALSE;
		ShowBox3 := FALSE;
	END_IF
	// Case commands: determine case position
	IF (ROSCommand.IntentName = 'caseLocator') THEN
		IF (ROSCommand.Slot[0].Value = 'Blue') THEN
			IF (ShowBox1) THEN
				textCommand := 'The blue case is ';
				brsftoa(BoxPosition1,ADR(TempString));
				brsstrcat(ADR(textCommand),ADR(TempString));
				brsstrcat(ADR(textCommand),ADR(' meters away from the infeed.'));
				speakNow := TRUE;
			ELSE
				textCommand := 'The blue case is not present.';
				speakNow := TRUE;
			END_IF
		ELSIF (ROSCommand.Slot[0].Value = 'Green') THEN
			IF (ShowBox2) THEN
				textCommand := 'The green case is ';
				brsftoa(BoxPosition2,ADR(TempString));
				brsstrcat(ADR(textCommand),ADR(TempString));
				brsstrcat(ADR(textCommand),ADR(' meters away from the infeed.'));
				speakNow := TRUE;
			ELSE
				textCommand := 'The green case is not present.';
				speakNow := TRUE;
			END_IF
		ELSIF (ROSCommand.Slot[0].Value = 'red') THEN
			IF (ShowBox3) THEN
				textCommand := 'The red case is ';
				brsftoa(BoxPosition3,ADR(TempString));
				brsstrcat(ADR(textCommand),ADR(TempString));
				brsstrcat(ADR(textCommand),ADR(' meters away from the infeed.'));
				speakNow := TRUE;
			ELSE
				textCommand := 'The red case is not present.';
				speakNow := TRUE;
			END_IF
		END_IF
	END_IF

	// Notification prompt for photoeye
	IF (ROSCommand.IntentName = 'notificationPrompt') THEN
		IF (ROSCommand.Slot[0].Value = 'Blue') THEN
			NotifyBox1 := TRUE;
		ELSIF (ROSCommand.Slot[0].Value = 'Green') THEN
			NotifyBox2 := TRUE;
		ELSIF (ROSCommand.Slot[0].Value = 'red') THEN
			NotifyBox3 := TRUE;
		END_IF
	END_IF

	// Data retrieval command
	IF (ROSCommand.IntentName = 'speedLocator') THEN
		IF (Conveyor.Velocity = 0) THEN
			textCommand := 'The conveyor is not currently moving.';
		ELSE
			textCommand := 'The current conveyor speed is ';
			brsftoa(Conveyor.Velocity,ADR(TempString));
			brsstrcat(ADR(textCommand),ADR(TempString));
			brsstrcat(ADR(textCommand),ADR(' meters per second.'));
		END_IF
		speakNow := TRUE;
	END_IF
	brsmemset(ADR(ROSCommand),0,SIZEOF(ROSCommand));

	// Delayed speech actions
	IF ((NotifyBox1) AND (BoxPosition1 > NOTIFY_POSITION)) THEN
		NotifyBox1 := FALSE;
		textCommand := 'The blue case has passed the photo eye.';
		speakNow := TRUE;
	END_IF
	IF ((NotifyBox2) AND (BoxPosition2 > NOTIFY_POSITION)) THEN
		NotifyBox2 := FALSE;
		textCommand := 'The green case has passed the photo eye.';
		speakNow := TRUE;
	END_IF
	IF ((NotifyBox3) AND (BoxPosition3 > NOTIFY_POSITION)) THEN
		NotifyBox3 := FALSE;
		textCommand := 'The red case has passed the photo eye.';
		speakNow := TRUE;
	END_IF

END_ACTION
```

### Program Logical/Programs/ros (ANSIC)

#### Main.cpp - Init, cyclic, exit code
```cpp
#include <bur/plctypes.h>

#ifdef _DEFAULT_INCLUDES
	#include <AsDefault.h>
#endif

#include "hardware.h"
#include "ros/node_handle.h"
#include "std_msgs/String.h"
#include "std_msgs/Float64.h"
#include "voice_interaction_robot_msgs/FulfilledVoiceCommand.h"
#include "sensor_msgs/JointState.h"

// amount of memory to be allocated for heap storage must be specified for every ANSI C++ program with the bur_heap_size variable
unsigned long bur_heap_size = 0xFFFF;

// Message callback for the joint1State subscription
void jointCallback( const sensor_msgs::JointState& jointData)
{
	joint1ActualPosition = (REAL) jointData.position[0];
	joint2ActualPosition = (REAL) jointData.position[1];
	return;
}

// Create the node handle
ros::NodeHandle_<Hardware> nh;

//************** Handling the float64 messages *********************//
// Create the message objects
std_msgs::Float64 joint1Position;
// Create the publishers
ros::Publisher joint1Publisher("/rrbot/joint1_position_controller/command", &joint1Position);

//************** Handling the joint state messages *********************//
// Create my subscribers
ros::Subscriber<sensor_msgs::JointState> jointStates("/rrbot/joint_states", jointCallback);

void _INIT ProgramInit(void)
{
	nh.initNode();
	nh.subscribe(jointStates);
	nh.advertise(joint1Publisher);
}

void _CYCLIC ProgramCyclic(void)
{
	joint1Position.data = (float)joint1SetPosition;
	joint1Publisher.publish( &joint1Position);

	nh.spinOnce();
}

void _EXIT ProgramExit(void)
{
	// Insert code here
}
```

#### hardware.h
```c
#include <bur/plctypes.h>

#ifdef _DEFAULT_INCLUDES
#include <AsDefault.h>
#endif

class Hardware
{
	public:
	Hardware()
	{
		// Initializing all variables (otherwise they can have random values)
		_programStartTime = clock_ms();
		_step = 0;
		_ident = 0;
		_recvData = 0;
		_lastError = 0;
		_errorFlag = false;
		_recvTimeout = 0;
		brsmemset(reinterpret_cast<UDINT>(&_tcpOpen),0,sizeof(_tcpOpen));
		brsmemset(reinterpret_cast<UDINT>(&_tcpClient),0,sizeof(_tcpClient));
		brsmemset(reinterpret_cast<UDINT>(&_tcpRecv),0,sizeof(_tcpRecv));
		brsmemset(reinterpret_cast<UDINT>(&_tcpSend),0,sizeof(_tcpSend));
		brsmemset(reinterpret_cast<UDINT>(&_tcpClose),0,sizeof(_tcpClose));
	}

	// any initialization code necessary to use the serial port
	void init()
	{
		// we need to stay in this method until we've successfully connected, hence the while loop
		while (_step < 3) // STEP_CONNECTED
		{
			switch (_step)
			{
				case 0: // STEP_START
					initData();
					_step = 1; // STEP_OPEN_SOCKET
					break;

				/* opens ethernet interface for use with SSL */
				case 1: // STEP_OPEN_SOCKET
					openSocket();
					break;

				/* connects to the server */
				case 2: // STEP_CONNECT_TO_SERVER
					connectToServer();
					break;

				/* holding state once we're connected */
				case 3: // STEP_CONNECTED
					break;
			}
		}
	}

	// read a byte from the serial port. -1 = failure
	int read()
	{
		return receiveData();
	}

	// write data to the connection to ROS
	void write(USINT* data, int length)
	{
		sendData(data, length);
	}

	// returns milliseconds since start of program
	unsigned long time()
	{
		return (long) DiffT(clock_ms(),_programStartTime);
	}

	UDINT getLoopCounter()
	{
		return _loopCounter;
	}

	private:

	void initData()
	{
		/***** internal parameter assignments for all FBs *****/
		// TCP open FB
		_tcpOpen.pIfAddr 	= 0;
		_tcpOpen.port 		= 0;
		_tcpOpen.options 	= tcpOPT_REUSEADDR;

		// TCP client FB
		_tcpClient.portserv = 11411;
		_tcpClient.pServer  = (UDINT) "192.168.56.101";

		// TCP receive FB
		_tcpRecv.pData   = (UDINT) &(_recvData);
		_tcpRecv.datamax = sizeof(_recvData);
		_tcpRecv.flags   = 0;

		// TCP send FB
		_tcpSend.flags   = 0;
	}

	/* Opens a socket with the given port. */
	void openSocket()
	{
		_tcpOpen.enable = 1;

		TcpOpen(&_tcpOpen);

		if (_tcpOpen.status == ERR_OK)
		{
			_step 	  = 2; // STEP_CONNECT_TO_SERVER
			_ident 	  = _tcpOpen.ident;
		}
		else if (_tcpOpen.status != ERR_FUB_BUSY )
		{
			_step	  = 500; // STEP_ERROR
			_lastError = _tcpOpen.status;
		}
	}

	/* Connects to the given server. */
	void connectToServer()
	{
		_tcpClient.enable   = 1;
		_tcpClient.ident 	  = _ident;
		TcpClient(&_tcpClient);

		if (_tcpClient.status == ERR_OK)
		{
			_step = 3; // STEP_CONNECTED
		}
		else if (_tcpClient.status != ERR_FUB_BUSY)
		{
			_errorFlag = true;
			_step 	  = 6; // STEP_CLOSE_SOCKET
			_lastError = _tcpClient.status;
		}
	}

	/* Receives data from server. */
	INT receiveData()
	{
//		if (!_tcpRecv.enable)
//			_recvCounter = 0;
		_tcpRecv.enable  = 1;
		_tcpRecv.ident   = _ident;
		while ((_tcpRecv.status == ERR_FUB_ENABLE_FALSE) || (_tcpRecv.status == ERR_FUB_BUSY))
		{
			_recvCounter = _recvCounter + 1;
			TcpRecv(&_tcpRecv);
		}

		if (_tcpRecv.status == ERR_OK)
		{
			_recvTimeout = 0;
			_tcpRecv.enable = false;
			TcpRecv(&_tcpRecv);
			return _recvData;
		}
		else if (_tcpRecv.status == tcpERR_NO_DATA) 					/* no data received - try again */
		{
			_recvTimeout 	   = _recvTimeout + 1;
			_tcpRecv.enable = false;
			TcpRecv(&_tcpRecv);
			return -1;
		}
		else if (_tcpRecv.status == ERR_FUB_BUSY)
		{
			return -1;
		}
		else // we have an error
		{
			_errorFlag = true;
			_step 	  = 6; // STEP_CLOSE_SOCKET
			_lastError = _tcpSend.status;
			_tcpRecv.enable = false;
			TcpRecv(&_tcpRecv);
			return -1;
		}
	}

	/* Sends data to the server */
	void sendData(USINT* data, int length)
	{
		_tcpSend.enable  = 1;
		_tcpSend.ident   = _ident;
		_tcpSend.pData   = (UDINT) data;
		_tcpSend.datalen = (UDINT) length;
		TcpSend(&_tcpSend);
		while ((_tcpSend.status == ERR_FUB_BUSY) || (_tcpSend.status == ERR_FUB_ENABLE_FALSE))
		{
			TcpSend(&_tcpSend);
		}

		if (_tcpSend.status == ERR_OK)
		{
			_tcpSend.enable = false;
			TcpSend(&_tcpSend);
			_step = 5; // STEP_RECEIVE_DATA
			return;
		}
		else if (_tcpSend.status != ERR_FUB_BUSY)
		{
			_tcpSend.enable = false;
			TcpSend(&_tcpSend);
			_errorFlag = true;
			_step	  = 6; // STEP_CLOSE_SOCKET
			_lastError = _tcpSend.status;
			return;
		}
	}

	UDINT _programStartTime;
	UINT _step;
	UDINT _ident;
	USINT _recvData;
	UINT _lastError;
	BOOL _errorFlag;
	UDINT _recvTimeout;
	UDINT _loopCounter;
	UDINT _recvCounter;
	UDINT _sendCounter;
	TcpOpen_typ _tcpOpen;
	TcpClient_typ _tcpClient;
	TcpRecv_typ _tcpRecv;
	TcpSend_typ _tcpSend;
	TcpClose_typ _tcpClose;
};
```

#### Header.h
```c
#ifndef _ROS_std_msgs_Header_h
#define _ROS_std_msgs_Header_h

#include <stdint.h>
#include <string.h>
#include <stdlib.h>
#include "../ros/msg.h"
#include "../ros/time.h"

namespace std_msgs
{

  class Header : public ros::Msg
  {
    public:
      typedef uint32_t _seq_type;
      _seq_type seq;
      typedef ros::Time _stamp_type;
      _stamp_type stamp;
      typedef const char* _frame_id_type;
      _frame_id_type frame_id;

    Header():
      seq(0),
      stamp(),
      frame_id("")
    {
    }

    virtual int serialize(unsigned char *outbuffer) const
    {
      int offset = 0;
      *(outbuffer + offset + 0) = (this->seq >> (8 * 0)) & 0xFF;
      *(outbuffer + offset + 1) = (this->seq >> (8 * 1)) & 0xFF;
      *(outbuffer + offset + 2) = (this->seq >> (8 * 2)) & 0xFF;
      *(outbuffer + offset + 3) = (this->seq >> (8 * 3)) & 0xFF;
      offset += sizeof(this->seq);
      *(outbuffer + offset + 0) = (this->stamp.sec >> (8 * 0)) & 0xFF;
      *(outbuffer + offset + 1) = (this->stamp.sec >> (8 * 1)) & 0xFF;
      *(outbuffer + offset + 2) = (this->stamp.sec >> (8 * 2)) & 0xFF;
      *(outbuffer + offset + 3) = (this->stamp.sec >> (8 * 3)) & 0xFF;
      offset += sizeof(this->stamp.sec);
      *(outbuffer + offset + 0) = (this->stamp.nsec >> (8 * 0)) & 0xFF;
      *(outbuffer + offset + 1) = (this->stamp.nsec >> (8 * 1)) & 0xFF;
      *(outbuffer + offset + 2) = (this->stamp.nsec >> (8 * 2)) & 0xFF;
      *(outbuffer + offset + 3) = (this->stamp.nsec >> (8 * 3)) & 0xFF;
      offset += sizeof(this->stamp.nsec);
      uint32_t length_frame_id = strlen(this->frame_id);
      varToArr(outbuffer + offset, length_frame_id);
      offset += 4;
      memcpy(outbuffer + offset, this->frame_id, length_frame_id);
      offset += length_frame_id;
      return offset;
    }

    virtual int deserialize(unsigned char *inbuffer)
    {
      int offset = 0;
      this->seq =  ((uint32_t) (*(inbuffer + offset)));
      this->seq |= ((uint32_t) (*(inbuffer + offset + 1))) << (8 * 1);
      this->seq |= ((uint32_t) (*(inbuffer + offset + 2))) << (8 * 2);
      this->seq |= ((uint32_t) (*(inbuffer + offset + 3))) << (8 * 3);
      offset += sizeof(this->seq);
      this->stamp.sec =  ((uint32_t) (*(inbuffer + offset)));
      this->stamp.sec |= ((uint32_t) (*(inbuffer + offset + 1))) << (8 * 1);
      this->stamp.sec |= ((uint32_t) (*(inbuffer + offset + 2))) << (8 * 2);
      this->stamp.sec |= ((uint32_t) (*(inbuffer + offset + 3))) << (8 * 3);
      offset += sizeof(this->stamp.sec);
      this->stamp.nsec =  ((uint32_t) (*(inbuffer + offset)));
      this->stamp.nsec |= ((uint32_t) (*(inbuffer + offset + 1))) << (8 * 1);
      this->stamp.nsec |= ((uint32_t) (*(inbuffer + offset + 2))) << (8 * 2);
      this->stamp.nsec |= ((uint32_t) (*(inbuffer + offset + 3))) << (8 * 3);
      offset += sizeof(this->stamp.nsec);
      uint32_t length_frame_id;
      arrToVar(length_frame_id, (inbuffer + offset));
      offset += 4;
      for(unsigned int k= offset; k< offset+length_frame_id; ++k){
          inbuffer[k-1]=inbuffer[k];
      }
      inbuffer[offset+length_frame_id-1]=0;
      this->frame_id = (char *)(inbuffer + offset-1);
      offset += length_frame_id;
     return offset;
    }

    const char * getType(){ return "std_msgs/Header"; };
    const char * getMD5(){ return "2176decaecbce78abc3b96ef049fabed"; };

  };

}
#endif
```
